TYPE "UDT_CylDiag"
VERSION : 0.1
// -----------------------------------------------------------------------------
// Cylinder Diagnostic - Per-cylinder runtime snapshot
// Used as: DB_Diagnostic.CylDiag[1..8]  (indexed by cylinder number)
// Add new cylinders in OB1 without changing DB_Diagnostic.
// -----------------------------------------------------------------------------
   STRUCT
      State : Int;   // FB_CylinderControl state (-1=EStop 0=Idle 1=Ext... 10=Err)
      Pos : Real;   // Ruler position (mm); 0.0 if no analog sensor connected
      Sol_A : Bool;   // Solenoid A output (extend coil)
      Sol_B : Bool;   // Solenoid B output (retract coil)
      Error : Bool;   // Active error flag
      ErrorID : Word;   // Error code (16#05xx)
   END_STRUCT;

END_TYPE

TYPE "UDT_SpindleSnap"
VERSION : 0.1
// -----------------------------------------------------------------------------
// Spindle Diagnostic Snapshot - one entry in the spindle history ring buffer
// DB_Spindle.Hist_Log[0..19] stores the last 20 state-change events.
// A new entry is pushed whenever SpindleState, PrevStart, ReqStart or StartEdge
// changes value -- so the log captures every meaningful transition without
// flooding with identical scans.
// -----------------------------------------------------------------------------
   STRUCT
      Seq : Int;   // Rolling sequence number
      MachineState : Int;   // FB_Process.State
      State : Int;   // FB_SpindleControl state: 0=Idle 20=Running 30=Halt 999=Error
      ReqStart : Bool;   // FB_RecipeHandler.SpindleReqStart
      ReqStop : Bool;   // FB_RecipeHandler.SpindleReqStop
      bStart : Bool;   // FB_Process bSpindleStart
      bStop : Bool;   // FB_Process bSpindleStop
      StartInput : Bool;   // Composite Start pin at FB_SpindleControl
      StopInput : Bool;   // Composite Stop pin
      EnableIn : Bool;   // bDrivesEnable
      PrevStart : Bool;   // prevStart latch inside FB_SpindleControl
      StartEdge : Bool;   // Rising edge accepted by FB_SpindleControl
      MoveVelBusy : Bool;   // MC_MoveVelocity.Busy  -- TO accepted and processing command
      MoveVelInVel : Bool;   // MC_MoveVelocity.InVelocity -- motor at commanded speed
   END_STRUCT;

END_TYPE

TYPE "AlarmEntry"
VERSION : 0.1
// -----------------------------------------------------------------------------
// Alarm Entry for history
// -----------------------------------------------------------------------------
   STRUCT
      Timestamp {InstructionName := 'DTL'; LibVersion := '1.0'} : DTL;   // RD_SYS_T() at moment of alarm
      ErrorCode : Word;   // 16#xxxx error code
      ProgramNum : Int;   // Active recipe program at fault time (0 = none)
      LineNum : Int;   // Active recipe line at fault time (-1 = outside recipe)
      ErrorText : String[40];   // ITEM-26: English error text snapshot (first 40 chars of DB_HMI.ErrorText)
   END_STRUCT;

END_TYPE

DATA_BLOCK "DB_Error"
{ S7_Optimized_Access := 'TRUE' }
VERSION : 0.1
NON_RETAIN
// DB_ErrorCodes removed -- error codes are used as inline hex constants.
// Severity: 0=info, 1=warn, 2=error, 3=fatal
// -----------------------------------------------------------------------------
// DB_Error - Centralized error snapshot for debugging (non-invasive to HMI)
// -----------------------------------------------------------------------------
   VAR
      Active : Bool;   // TRUE when an active error is present
      Code : Word;   // Error code (matches DB_ErrorCodes)
      Severity : Byte;   // Priority tier: 1=warning, 2=project, 3=motion/TO, 4=safety (higher preempts lower on HMI display)
      Source : String[20];   // Originating FB or category (e.g. 'Recipe', 'Safety')
      Line : Int;   // Recipe line (if applicable) or -1
      TimeStamp {InstructionName := 'DTL'; LibVersion := '1.0'} : DTL;   // Timestamp captured with RD_SYS_T
      Details : String[120];   // Free text details / ActiveErrorText History ring buffer (last 10 errors) for post-mortem analysis
      History_Code : Array[1..10] of Word;
      History_Time {InstructionName := 'DTL'; LibVersion := '1.0'} : Array[1..10] of DTL;
      History_Source : Array[1..10] of String[20];
      History_Details : Array[1..10] of String[80];
      History_Index : Int;   // 1..10
      History_Count : Int;   // Number of valid entries (<=10)
      TotalErrorCount : DInt;   // Lifetime error count (incremented on each new error)
   END_VAR


BEGIN
   Active := FALSE;
   Code := 0;
   Severity := 0;
   Line := -1;
   History_Index := 0;
   History_Count := 0;
   TotalErrorCount := 0;

END_DATA_BLOCK

FUNCTION_BLOCK "FB_Axis_RelPos"
{ S7_Optimized_Access := 'TRUE' }
VERSION : 0.1
// =============================================================================
// FB_Axis_RelPos -- Relative position move (MC_MoveRelative wrapper)
//
// Unlike MC_MoveAbsolute, does not require homing.
// Distance: positive = forward, negative = backward.
// =============================================================================
   VAR_INPUT
      Execute : Bool;
      Distance : Real;   // Relative distance (mm or degrees)
      Velocity : Real;
   END_VAR

   VAR_OUTPUT
      Done : Bool;
      Busy : Bool;
      Error : Bool;
      ErrorID : Word;   // TO error code (MC_MoveRelative.ErrorID)
   END_VAR

   VAR_IN_OUT
      Axis {InstructionName := 'TO_PositioningAxis'; LibVersion := '8.0'} : TO_PositioningAxis;
   END_VAR

   VAR
      MC_MoveRelative_Instance {InstructionName := 'MC_MoveRelative'; LibVersion := '8.0'} : MC_MoveRelative;
      execLatch : Bool;
      prevExec : Bool;
      doneLatch : Bool;
   END_VAR


BEGIN

	IF #Execute AND NOT #prevExec THEN
	    #doneLatch := FALSE;
	    #execLatch := TRUE;
	END_IF;
	#prevExec := #Execute;

	#MC_MoveRelative_Instance(
	                          Axis := #Axis,
	                          Execute := #execLatch,
	                          Distance := #Distance,
	                          Velocity := #Velocity,
	                          Done => #Done,
	                          Busy => #Busy,
	                          Error => #Error
	);
	#ErrorID := #MC_MoveRelative_Instance.ErrorID;

	IF #MC_MoveRelative_Instance.Done OR #MC_MoveRelative_Instance.Error THEN
	    #execLatch := FALSE;
	    #doneLatch := TRUE;
	END_IF;

END_FUNCTION_BLOCK

FUNCTION_BLOCK "FB_Axis_Jog"
{ S7_Optimized_Access := 'TRUE' }
VERSION : 0.1
// =============================================================================
// FB_Axis_Jog -- Continuous jog move
//
// JogForward and JogBackward are level inputs (not edge).
// Axis decelerates when button is released.
// Velocity: jog speed (mm/s) -- fed from DB_Manual.JogSpeed.
// =============================================================================
   VAR_INPUT
      JogForward : Bool;   // Continuous jog in positive direction (level)
      JogBackward : Bool;   // Continuous jog in negative direction (level)
      Velocity : Real;   // Jog speed (mm/s)
   END_VAR

   VAR_OUTPUT
      Busy : Bool;
      Error : Bool;
   END_VAR

   VAR_IN_OUT
      Axis {InstructionName := 'TO_PositioningAxis'; LibVersion := '8.0'} : TO_PositioningAxis;
   END_VAR

   VAR
      MC_MoveJog_Instance {InstructionName := 'MC_MoveJog'; LibVersion := '8.0'} : MC_MoveJog;
   END_VAR


BEGIN

	#MC_MoveJog_Instance(
	                     Axis := #Axis,
	                     JogForward := #JogForward,
	                     JogBackward := #JogBackward,
	                     Velocity := #Velocity,
	                     Busy => #Busy,
	                     Error => #Error
	);

END_FUNCTION_BLOCK

DATA_BLOCK "DB_AlarmHistory"
{ S7_Optimized_Access := 'TRUE' }
VERSION : 0.1
NON_RETAIN
// -----------------------------------------------------------------------------
// DB_AlarmHistory - 20-entry alarm ring buffer for HMI history table (ITEM-26)
// NON_RETAIN: cleared on PLC power cycle. Survives Cmd_Reset (soft reset).
// HMI: connect Hist_Log[0..19] to a table, poll Hist_SeqNum for change detection,
//      sort by Timestamp descending. Hist_Clear = TRUE wipes manually.
// -----------------------------------------------------------------------------
   VAR
      Hist_Head : Int;   // Next write slot (0..19, wraps on overflow)
      Hist_Count : Int;   // Number of valid entries (0..20)
      Hist_SeqNum : DInt;   // Monotonically increasing â€” HMI polls for change detection
      Hist_Clear : Bool;   // HMI writes TRUE to clear history; auto-resets next scan
      Hist_Log : Array[0..19] of "AlarmEntry";
   END_VAR


BEGIN
   Hist_Head := 0;
   Hist_Count := 0;
   Hist_SeqNum := 0;
   Hist_Clear := FALSE;

END_DATA_BLOCK

DATA_BLOCK "DB_HMI_Errors"
{ S7_Optimized_Access := 'TRUE' }
VERSION : 0.1
NON_RETAIN
// -----------------------------------------------------------------------------
// DB_HMI_Errors - Error bits + Word triggers for HMI Alarm View
// -----------------------------------------------------------------------------
// Alarm Words (for HMI Discrete Alarm view)
   VAR
      AlarmWord_Axis : Word;
      AlarmWord_Limits : Word;
      AlarmWord_Tool : Word;
      AlarmWord_Recipe : Word;
      AlarmWord_Safety : Word;
      AlarmWord_Spindle : Word;
      AlarmWord_TO : Word;   // Individual Bool flags
      Err_X_MoveFailed : Bool;
      Err_Z_MoveFailed : Bool;
      Err_X_HomingFailed : Bool;
      Err_Z_HomingFailed : Bool;
      Err_DriveFault : Bool;
      Err_ToolDrivePower : Bool;   // ITEM-29: tool axis drive power fault (error code 0x000D)
      Err_ToolMoveFailed : Bool;
      Err_ToolHomingFailed : Bool;
      Err_MotionTimeout : Bool;
      Err_LockExtendTimeout : Bool;   // 16#0012 -- ToolHeadLock did not confirm engaged within timeout
      Err_SoftLimit_X_Min : Bool;
      Err_SoftLimit_X_Max : Bool;
      Err_SoftLimit_Z_Min : Bool;
      Err_SoftLimit_Z_Max : Bool;
      Err_HWLimit_X_Min : Bool;
      Err_HWLimit_X_Max : Bool;
      Err_HWLimit_Z_Min : Bool;
      Err_HWLimit_Z_Max : Bool;
      Err_InvalidToolNum : Bool;
      Err_ToolOutOfRange : Bool;
      Err_ToolRotTimeout : Bool;
      Err_ToolRetractFail : Bool;
      Err_ToolRotFailed : Bool;
      Err_Recipe_InvalidCmd : Bool;
      Err_Recipe_ParseErr : Bool;
      Err_Recipe_Empty : Bool;
      Err_Recipe_NoLines : Bool;
      Err_PreScan_Limits : Bool;
      Err_Recipe_Feedrate : Bool;
      Err_Recipe_Timeout : Bool;
      Err_Recipe_ToolNum : Bool;
      Err_EStop : Bool;
      Err_EStop_Discrepancy : Bool;   // E-Stop contact discrepancy (channel fault)
      Err_DoorOpen : Bool;
      Err_DrivesNotReady : Bool;
      Err_AirPressure : Bool;
      Err_SafetyInterlock : Bool;
      Err_Spindle_Power : Bool;
      Err_Spindle_Run : Bool;
      Err_Spindle_Halt : Bool;
      Err_Spindle_Speed : Bool;
      Err_TO_Position : Bool;
      Err_TO_Velocity : Bool;
      Err_TO_NotReady : Bool;
      Err_TO_NotEnabled : Bool;
      Err_TO_LimitExceeded : Bool;   // Summary flags
      AnyError : Bool;
      AnySafetyError : Bool;
      AnyAxisError : Bool;
      AnyLimitError : Bool;
      AnyToolError : Bool;
      AnyRecipeError : Bool;
      AnySpindleError : Bool;
   END_VAR


BEGIN

END_DATA_BLOCK

FUNCTION_BLOCK "FB_Axis_Home"
{ S7_Optimized_Access := 'TRUE' }
VERSION : 0.4
// =============================================================================
// FB_Axis_Home -- Homing
//
// Mode options (MC_Home Mode parameter):
//   0 -- Passive: only set current position to Position value
//   2 -- Active:  go to reference switch, zero encoder
//   3 -- Active + Zero: go to reference switch, set Position value
//
// Default mode = 3 (matches DB_Manual.HomingMode).
//
// Safety note: Execute is rising-edge triggered -- even if Execute stays TRUE
// after Done/Error, a new homing will not start. Same pattern as FB_Axis_AbsPos.
// =============================================================================
   VAR_INPUT
      Execute : Bool;   // Rising edge = start homing
      Mode : Int := 3;   // Homing mode (0=Passive, 2=Active, 3=Active+Zero)
      Position : Real := 0.0;   // Position value after homing (usually 0.0)
   END_VAR

   VAR_OUTPUT
      Done : Bool;
      Busy : Bool;
      Error : Bool;
      ErrorID : Word;   // MC_Home TO error code -- converted to readable text via FC_TO_ErrorText
   END_VAR

   VAR_IN_OUT
      Axis {InstructionName := 'TO_PositioningAxis'; LibVersion := '8.0'} : TO_PositioningAxis;
   END_VAR

   VAR
      MC_Home_Instance {InstructionName := 'MC_Home'; LibVersion := '8.0'} : MC_Home;
      execInternal : Bool;   // Actual Execute sent to MC_Home
      prevExecute : Bool;   // Previous Execute value for edge detection
      doneLatch : Bool;   // Prevents re-trigger after Done/Error
   END_VAR


BEGIN

	// Rising edge: new command -- clear doneLatch
	IF #Execute AND NOT #prevExecute THEN
	    #doneLatch := FALSE;
	END_IF;
	#prevExecute := #Execute;

	// execInternal: run if new command and not yet done, OR still busy
	// This ensures Execute staying TRUE after Done does not restart homing
	#execInternal := (#Execute AND NOT #doneLatch) OR #MC_Home_Instance.Busy;

	#MC_Home_Instance(
	                  Axis := #Axis,
	                  Execute := #execInternal,
	                  Position := #Position,
	                  Mode := #Mode,
	                  Done => #Done,
	                  Busy => #Busy,
	                  Error => #Error
	);

	// Done or Error: set doneLatch -- cannot re-trigger without Execute FALSEâ†’TRUE
	IF #MC_Home_Instance.Done OR #MC_Home_Instance.Error THEN
	    #doneLatch := TRUE;
	END_IF;

	// Pass TO error code out -- written to DB_Diagnostic in FB_Process
	#ErrorID := #MC_Home_Instance.ErrorID;

END_FUNCTION_BLOCK

TYPE "RecipeHeader"
VERSION : 0.1
   STRUCT
      sName : String[20];   // Program name (max 20 chars)
      LineCount : Int;   // Total lines in program (0-999)
      Valid : Bool;   // Program is valid and loaded
      PreScanned : Bool;   // Pre-scan completed
      MinX : Real;   // Bounding box Min X
      MaxX : Real;   // Bounding box Max X
      MinZ : Real;   // Bounding box Min Z
      MaxZ : Real;   // Bounding box Max Z
   END_STRUCT;

END_TYPE

DATA_BLOCK "DB_ToolConfig"
{ S7_Optimized_Access := 'TRUE' }
VERSION : 0.2
NON_RETAIN
// -----------------------------------------------------------------------------
// DB_ToolConfig - Tool changer configuration
// -----------------------------------------------------------------------------
// Slot angles -- automatically calculated by FC_ToolAngleCalc (AutoCalcAngles=TRUE)
// or manually entered from HMI Tool page (AutoCalcAngles=FALSE).
   VAR
      Tool1_Position : Real;   // Slot 1 angle (degrees)
      Tool2_Position : Real;   // Slot 2 angle (degrees)
      Tool3_Position : Real;   // Slot 3 angle (degrees)
      Tool4_Position : Real;   // Slot 4 angle (degrees) Slot code mapping -- can be entered from HMI Tool page. Operator enters which head code is in which slot.
      ToolCode_List : Array[1..4] of Int;
      CurrentTool : Int;   // Active slot number (1-4) HMI Tool page: automatic angle calculation TRUE = calculate evenly spaced based on ToolCount (e.g. 4 slots â†’ 0/90/180/270) FALSE = Tool1..4_Position open for manual entry
      AutoCalcAngles : Bool;   // Calculated step angle -- displayed on HMI for information (e.g. "90Â°/slot")
      ToolStepAngle_Calc : Real;
   END_VAR


BEGIN
   Tool1_Position := 0.0;
   Tool2_Position := 120.0;
   Tool3_Position := 240.0;
   Tool4_Position := 360.0;
   ToolCode_List[1] := 101;
   ToolCode_List[2] := 102;
   ToolCode_List[3] := 103;
   ToolCode_List[4] := 104;
   CurrentTool := 1;
   AutoCalcAngles := TRUE;
   ToolStepAngle_Calc := 120.0;

END_DATA_BLOCK

DATA_BLOCK "DB_MachineConfig"
{ S7_Optimized_Access := 'TRUE' }
VERSION : 0.2
NON_RETAIN
// -----------------------------------------------------------------------------
// DB_MachineConfig - Machine configuration parameters
// -----------------------------------------------------------------------------
// =====================================================================
// HMI-EDITABLE: Machine Physical Limits (mm)
// These values are NOT overwritten by FC_LoadConfig.
// Can be changed from HMI Setup screen; preserved on PLC restart.
// =====================================================================
   VAR
      SoftLimit_MinX : Real;   // X minimum (home=0)
      SoftLimit_MaxX : Real;   // X maximum travel (mm)
      SoftLimit_MinZ : Real;   // Z minimum (negative = mandrel front / clearance)
      SoftLimit_MaxZ : Real;   // Z maximum (forming depth) HMI-EDITABLE: Safe Positions (mm)
      SafePos_X : Real;   // "Go Safe" X target
      SafePos_Z : Real;   // "Go Safe" Z target (clearance zone) HMI-EDITABLE: Pause Retract (mm / mm/s) On Pause, X and Z jog by these signed offsets to pull the tool clear (spindle keeps running). On Continue they return to the exact interruption point before the recipe resumes. Retract target is clamped to soft limits. Offset 0 = that axis does not move on pause. See docs/Pause_Retract_Plan.md.
      PauseRetract_X : Real;   // Pause retract offset X (signed, mm)
      PauseRetract_Z : Real;   // Pause retract offset Z (signed, mm)
      PauseRetract_Vel : Real;   // Retract/return velocity (mm/s) HMI-EDITABLE: Homing Parameters
      HomeOffset_X : Real;   // X set value after homing
      HomeOffset_Z : Real;   // Z set value after homing
      HomeVelocity : Real;   // Homing clearance velocity (mm/s)
      PostHome_Clearance : Real;   // Distance to clear PNP zone after homing (mm)
      AlwaysHomeOnAutoStart : Bool;   // TRUE = home all axes on every auto start (recommended) âš ï¸ UNUSED: The following two parameters are not read anywhere in PLC code. Recipe handler takes its own feedrate from the recipe line. Do not connect to HMI. May be used if manual tool change sequence is added later.
      ToolChangePos_X : Real;   // (Unused) Safe X for manual tool change
      ToolChangePos_Z : Real;   // (Unused) Safe Z for manual tool change
      DefaultFeedrate : Real;   // (Unused) Default feedrate ===================================================================== FIXED: Hardware/TO Limits -- must not be changed from HMI FC_LoadConfig (OB100) writes these values on every restart. =====================================================================
      MaxVelocity : Real;   // mm/s - TO max velocity
      RapidVelocity : Real;   // mm/s - G0 rapid speed
      MinVelocity : Real;   // mm/s - TO minimum
      FeedrateConvFactor : Real;   // divisor to convert recipe F (mm/min) to axis velocity (mm/s) Tool Configuration -- HMI-EDITABLE: active slot count (1-4)
      ToolCount : Int;
      ToolVelocity : Real;   // deg/s -- turret rotation speed (clamped by TO max) Hardware configuration -- set TRUE if this axis is not physically connected to the machine (different from HMI bypasses: this is a hardware presence flag)
      Bypass_ToolAxis : Bool;
      Bypass_MandrelLock : Bool;   // Spindle deceleration wait: time between RunCmd=FALSE and next RunCmd=TRUE. Set to match VFD deceleration ramp time. HMI-editable.
      SpindleDecelTime : Time;   // Proportional MandrelLock release wait (ITEM-28). SpindleStopSafeTime = full-speed stop safety margin (tune to measured VFD decel time + margin). Formula: PT = (capturedRPM / SpindleMaxRPM) * SpindleStopSafeTime
      SpindleMaxRPM : Real;   // RPM -- denominator for proportional wait (match DB_Spindle.MaxSpeed)
      SpindleStopSafeTime : Time;   // Full-speed decel safety margin (tune on-site) â”€â”€â”€ Cylinder stroke wait times (open-loop: tuned to physical stroke duration) These are deliberate waits with no sensor feedback. Set slightly above measured stroke time.
      CylMandrelLock_ClampTime : Time;   // STATE_SHEET_WAIT ph.2: MandrelLock clamp stroke
      CylSheetHolder_RetractTime : Time;   // STATE_SHEET_WAIT ph.3: SheetHolder retract stroke
      CylToolHeadLock_PreDelay : Time;   // STATE_LOCK_EXTEND_WAIT: pre-delay before solenoid energises
      CylToolHeadLock_RetractTime : Time;   // STATE_LOCK_RETRACT_WAIT: spring-return wait (no sensor) â”€â”€â”€ Process timeouts (trigger errors when limits exceeded)
      Timeout_DriveReady : Time;   // STATE_STARTING: drives not ready within this time â†’ error
      Timeout_Homing : Time;   // STATE_HOMING + STATE_STOP_GOHOME combined timeout
      Timeout_Motion : Time;   // Per-line G0/G1 motion timeout in FB_RecipeHandler
      Timeout_SpindleAtSpeed : Time;   // CMD=20: spindle must reach target speed within this time
      Timeout_SpindleStop : Time;   // CMD=21: spindle must reach zero within this time
      Timeout_ToolChange : Time;   // Turret rotation must complete within this time
      Timeout_EStopDiscrep : Time;   // E-Stop dual-channel discrepancy debounce
   END_VAR


BEGIN
   SoftLimit_MinX := -10.0;
   SoftLimit_MaxX := 500.0;
   SoftLimit_MinZ := -10.0;
   SoftLimit_MaxZ := 500.0;
   SafePos_X := 0.0;
   SafePos_Z := 0.0;
   PauseRetract_X := -10.0;
   PauseRetract_Z := -10.0;
   PauseRetract_Vel := 30.0;
   HomeOffset_X := 0.0;
   HomeOffset_Z := 0.0;
   HomeVelocity := 10.0;
   PostHome_Clearance := 10.0;
   AlwaysHomeOnAutoStart := TRUE;
   ToolChangePos_X := 0.0;
   ToolChangePos_Z := 0.0;
   DefaultFeedrate := 100.0;
   MaxVelocity := 40.0;
   RapidVelocity := 40.0;
   MinVelocity := 1.0;
   FeedrateConvFactor := 60.0;
   ToolCount := 3;
   ToolVelocity := 50.0;
   Bypass_ToolAxis := FALSE;
   Bypass_MandrelLock := FALSE;
   SpindleDecelTime := T#2S;
   SpindleMaxRPM := 2400.0;
   SpindleStopSafeTime := T#20S;
   CylMandrelLock_ClampTime := T#5S;
   CylSheetHolder_RetractTime := T#5S;
   CylToolHeadLock_PreDelay := T#1S;
   CylToolHeadLock_RetractTime := T#3S;
   Timeout_DriveReady := T#3S;
   Timeout_Homing := T#2M;
   Timeout_Motion := T#5M;
   Timeout_SpindleAtSpeed := T#10S;
   Timeout_SpindleStop := T#15S;
   Timeout_ToolChange := T#30S;
   Timeout_EStopDiscrep := T#500MS;

END_DATA_BLOCK

FUNCTION_BLOCK "FB_Axis_Halt"
{ S7_Optimized_Access := 'TRUE' }
VERSION : 0.2
// =============================================================================
// FB_Axis_Halt -- Controlled stop
//
// Execute = TRUE â†’ MC_Halt called, axis decelerates to a stop.
// Cancels any active MC_MoveAbsolute.
// Done = TRUE â†’ axis has fully stopped.
// =============================================================================
   VAR_INPUT
      Execute : Bool;   // TRUE = issue stop command
   END_VAR

   VAR_OUTPUT
      Done : Bool;
      Busy : Bool;
      Error : Bool;
      ErrorID : Word;   // MC_Halt TO error code -- available for diagnostics on halt failure
   END_VAR

   VAR_IN_OUT
      Axis {InstructionName := 'TO_PositioningAxis'; LibVersion := '8.0'} : TO_PositioningAxis;
   END_VAR

   VAR
      MC_Halt_Instance {InstructionName := 'MC_Halt'; LibVersion := '8.0'} : MC_Halt;
   END_VAR


BEGIN

	#MC_Halt_Instance(
	                  Axis := #Axis,
	                  Execute := #Execute,
	                  Done => #Done,
	                  Busy => #Busy,
	                  Error => #Error,
	                  ErrorID => #ErrorID
	);

END_FUNCTION_BLOCK

TYPE "RecipeLine"
VERSION : 0.1
   STRUCT
      X : Real;   // 4 bytes - Target X position (mm)
      Z : Real;   // 4 bytes - Target Z position (mm)
      F : Int;   // 2 bytes - Feedrate (mm/min, 0=rapid)
      CMD : Byte;   // 1 byte  - Command: 0=G0, 1=G1, 10=Tool, 20=SpindleOn, 21=SpindleOff, 30=Dwell, 99=End
      Param : Byte;   // 1 byte  - CMD=10:ToolNum, CMD=20:RPM/10, CMD=30:Time*100ms
   END_STRUCT;

END_TYPE

DATA_BLOCK "DB_HMI"
{ S7_Optimized_Access := 'TRUE' }
VERSION : 0.3
NON_RETAIN
// =============================================================================
// 02_DataBlocks.scl
// All non-recipe data blocks.
// Recipe program DBs (DB_RecipeProgram1..5) are in 02b_RecipePrograms.scl.
// Target: CPU 1214C (100KB work memory)
// =============================================================================
// -----------------------------------------------------------------------------
// DB_HMI - Human Machine Interface data
// -----------------------------------------------------------------------------
// ===========================================================
// BUTTONS (Input) - Version_GCODE compatible
// ===========================================================
   VAR
      Btn_Start : Bool;   // Start machine
      Btn_Stop : Bool;   // Stop machine
      Btn_Pause : Bool;   // Pause/Resume toggle
      Btn_Reset : Bool;   // Reset program to beginning
      Btn_ApplyToolConfig : Bool;   // Apply tool-slot codes from HMI to DB_ToolConfig
      Btn_AckError : Bool;   // Acknowledge error â†’ transitions from STATE_ERROR to STOPPED
      Btn_Continue : Bool;   // Continue from pause (PAUSED) -- STATE_PAUSED â†’ RUNNING
      Btn_Restart : Bool;   // STATE_ERROR or PAUSED â†’ STOPPED (restart with Start)
      Btn_ProdReset : Bool;   // Reset production counters + history
      Btn_LastCycleReset : Bool;   // Reset last cycle summary only (counters preserved) NOTE: Btn_ProdReset already does this too. If not adding both as separate HMI buttons, Btn_LastCycleReset is redundant -- do not connect to HMI if unused. =========================================================== MODE SELECTION (Input) ===========================================================
      ProductSelect : Int;   // Recipe selector (1-5)
      FeedrateOverride : Real;   // Speed % for G1 moves (50-200, 100=normal)
      RapidOverride : Real;   // Speed % for G0 rapid moves (50-200)
      SingleStepMode : Bool;   // TRUE = stop after each line, wait for StepNext
      StepNext : Bool;   // Pulse to advance one step in SingleStepMode Program names and validity -- PLC does NOT write to these tags. Written by CAM post-processor or HMI operator. Can be read for displaying the program list on HMI.
      ProgramNames : Array[1..5] of String[20];   // Operator-defined program names
      ProgramValid : Array[1..5] of Bool;   // Is program loaded? (written by HMI/CAM) Tool slot codes editable from HMI. Enter external codes like 101, 406 etc. These are copied to DB_ToolConfig.ToolCode_List when operator presses Apply.
      ToolSlotCode : Array[1..4] of Int;   // =========================================================== POSITION DISPLAYS (Output) ===========================================================
      ActualX : Real;   // Current X position (mm)
      ActualZ : Real;   // Current Z position (mm) =========================================================== STATUS DISPLAYS (Output) ===========================================================
      StatusMsg : String[50];   // Status message text
      MachineState : Int;   // State machine state
      CurrentLine : Int;   // Current line being executed
      TotalLines : Int;   // Total lines in program
      ProgressPercent : Real;   // Progress 0-100%
      CurrentTool : Int;   // Active tool (1-4)
      FeedrateActive : Real;   // Actual feedrate (mm/min) âš ï¸ UNUSED: PLC code does not write to the Axis_Status_* tags below anywhere. They will always be 0 / empty if connected to HMI. Reserved for future use -- do not display on HMI for now.
      Axis_Status_X : Int;
      Axis_Status_Z : Int;
      Axis_Status_Spindle : Int;
      Axis_Status_Toolhead : Int;
      Axis_Status_X_Str : String[10];
      Axis_Status_Z_Str : String[10];
      Axis_Status_Spindle_Str : String[10];
      Axis_Status_Toolhead_Str : String[10];   // =========================================================== STATUS LAMPS (Output) ===========================================================
      IsRunning : Bool;   // Machine is running
      IsPaused : Bool;   // Machine is paused
      HasError : Bool;   // Error is active
      ElapsedTime : Time;   // Program elapsed time
      ElapsedSeconds : DInt;   // Elapsed time in seconds (for HMI display)
      CycleCount : Int;   // Number of completed programs =========================================================== ERROR DISPLAY (Output) ===========================================================
      ErrorID : Word;   // Error code (0=OK)
      ErrorText : String[100];   // Error description
      ErrorDetail : String[120];   // Additional error info =========================================================== WARNING DISPLAY (Output) ===========================================================
      HasWarning : Bool;   // TRUE when a non-blocking warning is active (E-Stop bypass or sheet insert prompt)
      WarningText : String[70];   // Warning message text -- English (E-Stop bypass or operator prompts only)
      ResumeLine : Int;   // Saved recipe line for warm restart (-1 = none). Set in STATE_ERROR, cleared on Btn_Restart. =========================================================== SPANISH TEXT MIRRORS (Output) -- for Mexican operator HMI PLC writes these every scan alongside the English equivalents. Connect to a second-language screen or a language-toggle switch. ===========================================================
      StatusMsg_ES : String[50];   // Estado actual (EspaÃ±ol)
      ErrorText_ES : String[100];   // Descripcion de error (EspaÃ±ol)
      ErrorDetail_ES : String[120];   // Detalle adicional (EspaÃ±ol)
      WarningText_ES : String[80];   // Advertencia (EspaÃ±ol) =========================================================== BYPASS SWITCHES (for testing) - Version_GCODE compatible âš ï¸ All bypasses reset to FALSE on restart (FC_LoadConfig). All must be FALSE in production. ===========================================================
      Bypass_EStop : Bool;   // Used in FB_SafetyMonitor âœ…
      Bypass_Door : Bool;   // Used in FB_SafetyMonitor âœ…
      Bypass_AirPressure : Bool;   // Used in FB_SafetyMonitor âœ…
      Bypass_Drives : Bool;   // Used in FB_SafetyMonitor âœ…
      Bypass_Spindle : Bool;   // Skips spindle commands in recipe (FB_RecipeHandler) -- dry run / commissioning
      Bypass_ToolChanger : Bool;   // âš ï¸ UNUSED -- not in safety monitor
      Bypass_MandrelLock : Bool;   // TRUE = machine variant without MandrelLock cylinder (manual clamping) =========================================================== BOUNDING BOX (Output - from pre-scan) ===========================================================
      BoundingBox_MinX : Real;
      BoundingBox_MaxX : Real;
      BoundingBox_MinZ : Real;
      BoundingBox_MaxZ : Real;
      BoundingBox_Valid : Bool;
      PreScanProgress : Real;   // Pre-scan progress 0-100% (written during STATE_PRE_SCAN) =========================================================== MANUAL > MANAGE: Contactor & Enable controls (Input) HMI writes these; PLC drives physical outputs in OB1. Buttons are toggles (maintained, not momentary). ===========================================================
      Btn_Contactor_X : Bool;   // Energize X driver contactor
      Btn_Contactor_Z : Bool;   // Energize Z driver contactor
      Btn_Contactor_Tool : Bool;   // Energize Tool driver contactor
      Btn_Contactor_Spindle : Bool;   // Energize Spindle driver contactor
      Btn_Enable_X : Bool;   // Send enable signal to X drive
      Btn_Enable_Z : Bool;   // Send enable signal to Z drive MANUAL > MANAGE: Status feedback (Output) for HMI lamps PLC writes these back after applying safety interlock.
      Contactor_X_On : Bool;
      Contactor_Z_On : Bool;
      Contactor_Tool_On : Bool;
      Contactor_Spindle_On : Bool;
      Enable_X_On : Bool;
      Enable_Z_On : Bool;   // =========================================================== E-STOP DUAL CHANNEL STATUS (Output - PLC writes, HMI reads) ===========================================================
      EStop_Ch1_OK : Bool;   // Channel 1 contact state (TRUE=closed=safe)
      EStop_Ch2_OK : Bool;   // Channel 2 contact state (TRUE=closed=safe)
      EStop_Discrepancy : Bool;   // Ch1 â‰  Ch2 â†’ contact fault, service required
   END_VAR


BEGIN
   ProductSelect := 1;
   FeedrateOverride := 100.0;
   RapidOverride := 100.0;
   SingleStepMode := FALSE;
   StepNext := FALSE;
   ToolSlotCode[1] := 101;
   ToolSlotCode[2] := 102;
   ToolSlotCode[3] := 103;
   ToolSlotCode[4] := 104;
   ResumeLine := -1;
   Bypass_EStop := FALSE;
   Bypass_Door := TRUE;
   Bypass_AirPressure := TRUE;
   Bypass_Drives := FALSE;
   Bypass_Spindle := FALSE;
   Bypass_ToolChanger := FALSE;
   Bypass_MandrelLock := FALSE;
   PreScanProgress := 0.0;

END_DATA_BLOCK

DATA_BLOCK "DB_Diagnostic"
{ S7_Optimized_Access := 'TRUE' }
VERSION : 0.1
NON_RETAIN
// -----------------------------------------------------------------------------
// DB_Diagnostic - Runtime diagnostics and debugging
// -----------------------------------------------------------------------------
// =========================================================
// PROCESS STATE
// =========================================================
   VAR
      Process_State : Int;
      Process_SafeToRun : Bool;
      Process_DrivesEnable : Bool;   // ========================================================= RECIPE HANDLER STATE =========================================================
      Recipe_CurrentProgram : Int;   // Active program number (1-5)
      Recipe_CurrentLine : Int;   // Current line being executed
      Recipe_TotalLines : Int;   // Total lines in program
      Recipe_TargetX : Real;   // Current target X
      Recipe_TargetZ : Real;   // Current target Z
      Recipe_Velocity : Real;   // Current velocity Pre-scan results
      PreScan_Complete : Bool;
      PreScan_Valid : Bool;   // No limit violations found
      PreScan_ErrorLine : Int;   // Line with limit error (-1 if none) ========================================================= MOVE STATUS =========================================================
      MoveX_Busy : Bool;
      MoveX_Done : Bool;
      MoveX_Error : Bool;
      MoveZ_Busy : Bool;
      MoveZ_Done : Bool;
      MoveZ_Error : Bool;
      bMoveX : Bool;   // X axis needs to move
      bMoveZ : Bool;   // Z axis needs to move ========================================================= AXIS INFO (commissioning) =========================================================
      Axis_X_Pos : Real;
      Axis_Z_Pos : Real;
      Axis_X_Enabled : Bool;
      Axis_Z_Enabled : Bool;
      Axis_X_Homed : Bool;
      Axis_Z_Homed : Bool;   // ========================================================= ERROR CONTEXT =========================================================
      Error_ProcessState : Int;
      Error_Line : Int;
      Error_Code : Word;   // TO error codes -- raw WORD codes from Siemens MC_ function blocks. Converted to readable text via FC_TO_ErrorText; compare with TIA Portal TO Diagnostics.
      MoveX_ErrorID : Word;   // MC_MoveAbsolute X axis TO code
      MoveZ_ErrorID : Word;   // MC_MoveAbsolute Z axis TO code
      HomeX_ErrorID : Word;   // MC_Home X axis TO code
      HomeZ_ErrorID : Word;   // MC_Home Z axis TO code
      HomeTool_ErrorID : Word;   // MC_Home Tool axis TO code
      Power_X_ErrorID : Word;   // MC_Power X axis TO code
      Power_Z_ErrorID : Word;   // MC_Power Z axis TO code
      Spindle_TO_ErrorID : Word;   // MC_Power/MC_MoveVelocity/MC_Halt spindle TO code
      Error_Text : String[100];   // Error_Detail removed -- not written anywhere, Error_Text is used instead Readable description for the last TO error code (FC_TO_ErrorText output)
      TO_ErrorText : String[60];   // ========================================================= CYLINDER DIAGNOSTICS -- indexed by cylinder number (1-based, max 8) No new fields needed when adding cylinders -- write to CylDiag[N] in OB1. =========================================================
      CylDiag : Array[1..8] of "UDT_CylDiag";
   END_VAR


BEGIN

END_DATA_BLOCK

DATA_BLOCK "DB_Spindle"
{ S7_Optimized_Access := 'TRUE' }
VERSION : 0.2
NON_RETAIN
// -----------------------------------------------------------------------------
// DB_Spindle - Spindle configuration and status
// -----------------------------------------------------------------------------
// Configuration
   VAR
      MinSpeed : Real;   // Minimum spindle speed (RPM)
      MaxSpeed : Real;   // Maximum spindle speed (RPM)
      DefaultSpeed : Real;   // Default spindle speed (RPM)
      SpeedTolerance : Real;   // Speed tolerance for AtSpeed (%)
      Bypass_AtSpeed : Bool;   // TRUE = skip AtSpeed wait (use during commissioning without drive) Commands (input from HMI/Program)
      Cmd_SetSpeed : Real;   // Commanded speed
      Cmd_Direction : Int;   // 1=CW, -1=CCW
      SpeedOverride : Real;   // Speed override (%) Status (output)
      IsRunning : Bool;
      AtSpeed : Bool;
      ActualSpeed : Real;
      CommandedSpeed : Real;
      Error : Bool;
      ErrorID : Word;   // ===================================================================== DIAGNOSTICS -- written every scan; read from HMI watch table Use these to trace the spindle start chain without TIA Portal online. Chain:  ReqStart â†’ bSpindleStart â†’ StartInput â†’ PrevStart â†’ StartEdge â†’ state =====================================================================
      Diag_SpindleState : Int;   // FB_SpindleControl state (0=Idle, 10=Starting, 20=Running, 30=Stopping, 999=Error)
      Diag_StartInput : Bool;   // Actual Start pin arriving at FB_SpindleControl (Manual OR bSpindleStart)
      Diag_StopInput : Bool;   // Actual Stop pin arriving at FB_SpindleControl
      Diag_EnableInput : Bool;   // Actual Enable pin (bDrivesEnable)
      Diag_StartEdge : Bool;   // Rising edge computed inside FB_SpindleControl (TRUE = spindle command accepted)
      Diag_PrevStart : Bool;   // prevStart latch inside FB_SpindleControl (must go FALSE between starts)
      Diag_bSpindleStart : Bool;   // FB_Process internal flag bSpindleStart (set by recipe or RUNNING state)
      Diag_bSpindleStop : Bool;   // FB_Process internal flag bSpindleStop
      Diag_ReqStart : Bool;
      Diag_ReqStop : Bool;
      Diag_MoveVelBusy : Bool;   // MC_MoveVelocity.Busy   -- TO is processing the velocity command
      Diag_MoveVelInVel : Bool;   // MC_MoveVelocity.InVelocity -- motor reached commanded speed ===================================================================== HISTORY RING BUFFER -- last 20 state-change snapshots A new entry is pushed whenever SpindleState, PrevStart, ReqStart or StartEdge changes, capturing every meaningful transition in sequence. How to read:   1. Hist_Count tells you how many valid entries exist (0..20).   2. Hist_Head-1 (mod 20) is the MOST RECENT entry.   3. Entries are indexed [0..19]; read them in Seq order.   4. Write Hist_Clear := TRUE from HMI to wipe and start fresh. =====================================================================
      Hist_Head : Int;   // Next write position (0..19, wraps)
      Hist_Count : Int;   // Number of valid entries (0..20)
      Hist_SeqNum : Int;   // Rolling sequence counter
      Hist_Clear : Bool;   // HMI: write TRUE to clear buffer (auto-resets)
      Hist_Log : Array[0..19] of "UDT_SpindleSnap";
   END_VAR


BEGIN
   MinSpeed := 120.0;
   MaxSpeed := 3000.0;
   DefaultSpeed := 1200.0;
   SpeedTolerance := 5.0;
   Bypass_AtSpeed := FALSE;
   SpeedOverride := 100.0;
   IsRunning := FALSE;
   AtSpeed := FALSE;
   ActualSpeed := 0.0;
   CommandedSpeed := 0.0;
   Error := FALSE;
   ErrorID := 0;
   Hist_Head := 0;
   Hist_Count := 0;
   Hist_SeqNum := 0;
   Hist_Clear := FALSE;

END_DATA_BLOCK

DATA_BLOCK "DB_SystemEvents"
{ S7_Optimized_Access := 'TRUE' }
VERSION : 0.2
NON_RETAIN
// =============================================================================
// Version_Recipe - 07_ReportError.scl
// Central helper to report errors from any FB/FC/FCU without duplicating logic.
// =============================================================================
// ---------------------------------------------------------------------------
// DB_SystemEvents - small DB for inter-block requests (error reporting)
// ---------------------------------------------------------------------------
// Error queue: ring buffer (4 slots) -- prevents silent loss when two errors
// occur in the same scan before FB_AlarmManager can consume the first entry.
// FC_ReportError enqueues; FB_AlarmManager dequeues one item per scan.
   VAR
      EQ_Head : Int;   // Next slot to dequeue (read index)
      EQ_Tail : Int;   // Next slot to enqueue (write index)
      EQ_Count : Int;   // Number of pending items (0..4)
      EQ_Code : Array[0..3] of Word;
      EQ_Details : Array[0..3] of String[80];
      EQ_Source : Array[0..3] of String[20];
   END_VAR


BEGIN
   EQ_Head := 0;
   EQ_Tail := 0;
   EQ_Count := 0;

END_DATA_BLOCK

FUNCTION_BLOCK "FB_Axis_AbsPos"
{ S7_Optimized_Access := 'TRUE' }
VERSION : 1.0
// =============================================================================
// 03_AxisControl.scl
// Axis control wrapper function blocks
//
// This file wraps Siemens PLCopen MC_ commands with project-specific thin wrappers.
// All FBs accept a TO_PositioningAxis VAR_IN_OUT reference.
//
// FB List:
//   FB_Axis_AbsPos  -- Absolute position move (MC_MoveAbsolute wrapper)
//   FB_Axis_Power   -- Drive enable/disable (MC_Power wrapper)
//   FB_Axis_Home    -- Homing (MC_Home wrapper)
//   FB_Axis_Halt    -- Controlled stop (MC_Halt wrapper)
//   FB_Axis_Jog     -- Continuous jog (MC_MoveJog wrapper)
//   FB_Axis_Reset   -- TO error reset (MC_Reset wrapper)
//
// Units: mm and mm/s (must match Technology Object configuration).
// =============================================================================
// =============================================================================
// FB_Axis_AbsPos -- Absolute position move
//
// Behavior:
//   Starts a new move on the rising edge of Execute.
//   Done = TRUE remains set while Execute is TRUE after completion.
//   Clearing Execute also clears Done -- ready for the next command.
//
// Usage note:
//   Used by FB_RecipeHandler and FB_ManualMode.
//   Two simultaneous Execute signals must not be sent to the same axis.
// =============================================================================
   VAR_INPUT
      Execute : Bool;   // Rising edge = new move command
      Position : Real;   // Target position (mm)
      Velocity : Real;   // Move velocity (mm/s)
   END_VAR

   VAR_OUTPUT
      Done : Bool;   // Move completed
      Busy : Bool;   // Move in progress
      Error : Bool;   // TO/drive error
      ErrorID : Word;   // MC_ error code (compare with TO diagnostics)
   END_VAR

   VAR_IN_OUT
      Axis {InstructionName := 'TO_PositioningAxis'; LibVersion := '8.0'} : TO_PositioningAxis;
   END_VAR

   VAR
      MC_MoveAbsolute_Instance {InstructionName := 'MC_MoveAbsolute'; LibVersion := '8.0'} : MC_MoveAbsolute;
      execLatch : Bool;   // MC_MoveAbsolute Execute latch -- ensures single command
      doneLatch : Bool;   // Holds Done result until Execute goes FALSE
      prevExecute : Bool;   // Previous Execute value for edge detection
   END_VAR


BEGIN

	// Rising edge: new command starting -- clear previous Done
	IF #Execute AND NOT #prevExecute THEN
	    #doneLatch := FALSE;
	END_IF;
	#prevExecute := #Execute;

	// If Execute is active, not yet done, and latch not set -- start move
	IF #Execute AND NOT #execLatch AND NOT #doneLatch THEN
	    #execLatch := TRUE;
	END_IF;

	// MC_MoveAbsolute call
	#MC_MoveAbsolute_Instance(
	                          Axis := #Axis,
	                          Execute := #execLatch,
	                          Position := #Position,
	                          Velocity := #Velocity,
	                          Done => #Done,
	                          Busy => #Busy,
	                          Error => #Error,
	                          ErrorID => #ErrorID
	);

	// Done: release latch, hold done result
	IF #MC_MoveAbsolute_Instance.Done THEN
	    #execLatch := FALSE;
	    #doneLatch := TRUE;
	    // Error or CommandAborted: release latch, do NOT set doneLatch
	    // CommandAborted happens when MC_Halt interrupts a running move (stop/pause/reset).
	    // Without this branch execLatch stays TRUE across recipe runs, MC never gets a new
	    // rising edge on Execute, and the axis stands still on the next start.
	ELSIF #MC_MoveAbsolute_Instance.Error OR #MC_MoveAbsolute_Instance.CommandAborted THEN
	    #execLatch := FALSE;
	END_IF;

	// Done: latch or MC instant done -- visible while Execute is TRUE
	#Done := #doneLatch OR #MC_MoveAbsolute_Instance.Done;
	#Error := #MC_MoveAbsolute_Instance.Error;

END_FUNCTION_BLOCK

FUNCTION_BLOCK "FB_InputManager"
{ S7_Optimized_Access := 'TRUE' }
VERSION : 1.0
// =============================================================================
// Version_Recipe - 06_MainProcess.scl
// Main process with recipe-based G-code and pre-scan validation
// =============================================================================
// -----------------------------------------------------------------------------
// FB_InputManager - OR-combine inputs from HMI, Panel, Remote
// DOC:
//  purpose: Create single rising-edge command outputs (Cmd_*) from multiple input sources.
//  inputs: HMI_*, Panel_*, Rem_* (Bool) - raw button states (level)
//  outputs: Cmd_* (Bool) - one-shot rising-edge commands for the system
//  notes: Uses prev* latches to detect rising edges; keeps logic simple for deterministic behavior.
// -----------------------------------------------------------------------------
   VAR_INPUT
      HMI_Start : Bool;   // HMI Start button (level)
      HMI_Stop : Bool;   // HMI Stop button (level)
      HMI_Pause : Bool;   // HMI Pause button (level)
      HMI_Reset : Bool;   // HMI Reset button (level)
      Panel_Start : Bool;   // Physical panel Start
      Panel_Stop : Bool;   // Physical panel Stop
      Panel_Pause : Bool;   // Physical panel Pause
      Panel_Reset : Bool;   // Physical panel Reset
      Rem_Start : Bool;   // Remote Start (e.g. PLC network)
      Rem_Stop : Bool;   // Remote Stop One-shot command outputs (rising edge true for one cycle)
   END_VAR

   VAR_OUTPUT
      Cmd_Start : Bool;
      Cmd_Stop : Bool;
      Cmd_Pause : Bool;
      Cmd_Reset : Bool;   // Previous sampled raw values for edge detection
   END_VAR

   VAR
      prevStart : Bool;
      prevStop : Bool;
      prevPause : Bool;
      prevReset : Bool;   // Combined raw inputs for current cycle
      rawStart : Bool;
      rawStop : Bool;
      rawPause : Bool;
      rawReset : Bool;
   END_VAR


BEGIN

	#rawStart := #HMI_Start OR #Panel_Start OR #Rem_Start;
	#rawStop := #HMI_Stop OR #Panel_Stop OR #Rem_Stop;
	#rawPause := #HMI_Pause OR #Panel_Pause;
	#rawReset := #HMI_Reset OR #Panel_Reset;
	#Cmd_Start := #rawStart AND NOT #prevStart;
	#Cmd_Stop := #rawStop AND NOT #prevStop;
	#Cmd_Pause := #rawPause AND NOT #prevPause;
	#Cmd_Reset := #rawReset AND NOT #prevReset;
	#prevStart := #rawStart;
	#prevStop := #rawStop;
	#prevPause := #rawPause;
	#prevReset := #rawReset;

END_FUNCTION_BLOCK

DATA_BLOCK "DB_RecipeProgram3"
{ S7_Optimized_Access := 'TRUE' }
VERSION : 0.1
NON_RETAIN
// -----------------------------------------------------------------------------
// DB_RecipeProgram3 - Recipe data for Program 3
// -----------------------------------------------------------------------------
   VAR
      Header : "RecipeHeader";
      Lines : Array[0..349] of "RecipeLine";
   END_VAR


BEGIN

END_DATA_BLOCK

DATA_BLOCK "DB_Manual"
{ S7_Optimized_Access := 'TRUE' }
VERSION : 0.3
NON_RETAIN
// -----------------------------------------------------------------------------
// DB_Manual - Manual mode control
// -----------------------------------------------------------------------------
   VAR
      ManualModeActive : Bool;
      SelectedAxis : Int;   // 0=X, 1=Z, 2=Tool, 3=Spindle
      ActiveAxis : Int;   // Currently active axis (-1 = none)
      JogSpeed : Real;   // mm/s
      JogIncrement : Real;   // mm per step
      HomingMode : Int;   // 0=Passive, 2=Active, 3=Active+Zero
      HomePosition : Real;   // Home position offset Jog buttons (both naming conventions)
      Btn_JogPlus : Bool;
      Btn_JogMinus : Bool;
      Jog_Plus : Bool;   // Alias
      Jog_Minus : Bool;   // Alias
      Btn_StepPlus : Bool;   // Incremental step +
      Btn_StepMinus : Bool;   // Incremental step - Homing buttons
      Btn_Home : Bool;
      Btn_HomeAxis : Bool;   // Alias for Btn_Home
      Btn_HomeAll : Bool;   // Home all axes
      Btn_GoSafe : Bool;
      Btn_GoZero : Bool;   // Absolute move
      MoveToPosition : Real;   // Target position
      Btn_MoveAbsolute : Bool;   // Execute move Tool step buttons
      Btn_ToolStepCW : Bool;   // Tool step clockwise
      Btn_ToolStepCCW : Bool;   // Tool step counter-clockwise
      ToolStepAngle : Real;   // Step angle (degrees)
      ToolStepSpeed : Real;   // Tool step velocity (deg/s)
      ToolPosition : Real;   // Current tool position (degrees) Spindle manual control
      Btn_SpindleStart : Bool;   // Start spindle
      Btn_SpindleStop : Bool;   // Stop spindle
      Btn_SpindleAckError : Bool;   // Acknowledge spindle error only (machine reset not required)
      Manual_SpindleSpeed : Real;   // Spindle speed (RPM)
      Manual_SpindleDir : Int;   // 1=CW, -1=CCW Status (multiple naming conventions for HMI compatibility)
      JogBusy : Bool;
      ManualBusy : Bool;   // Alias for JogBusy
      JogError : Bool;
      ManualError : Bool;   // Alias for JogError
      JogErrorID : Word;
      ManualErrorID : Word;   // Alias for JogErrorID Selected axis info (output)
      SelectedAxisName : String[20];
      SelectedAxisPos : Real;
      SelectedAxisHomed : Bool;
      SelectedAxisReady : Bool;   // =========================================================== CYLINDER MANUAL CONTROL One HMI screen controls all cylinders via SelectedCylinder. HMI writes to these fields; FC_CylinderDispatch routes to the correct DB_CylinderX instance each scan. To add a cylinder: add DB_CylinderN in 02_DataBlocks.scl, add OB1 calls, and add a CASE branch in FC_CylinderDispatch. ===========================================================
      SelectedCylinder : Int;   // Active cylinder (1..N)
      Btn_CylExtend : Bool;   // Extend command
      Btn_CylExtendFull : Bool;   // Full extend (ignore sensor)
      Btn_CylRetract : Bool;   // Retract command
      Btn_CylRetractFull : Bool;   // Full retract (bypass sensors, pulse use)
      Btn_CylGotoPos : Bool;   // Rising edge: go to target (Mode 2 = zone-pulse, Mode 3 = extend to level)
      Cyl_TargetPos : Real;   // [Modes 2+3] Target position (mm)
      Cyl_Tolerance : Real;   // [Mode 2] Tolerance written to cylinder DB on Btn_ApplyType press
      Btn_ApplyType : Bool;   // Rising edge: write SelCyl_SetType + Cyl_Tolerance â†’ cylinder DB
      SelCyl_SetType : Int;   // Desired PositioningMode (0â€“3) â€” HMI input field
      prevBtn_ApplyType : Bool;   // Edge detection (internal, not for HMI) Selected cylinder status (PLC â†’ HMI)
      SelCyl_Name : String[20];   // "Cylinder 1" etc.
      SelCyl_State : Int;   // State code
      SelCyl_StateText : String[14];   // State text
      SelCyl_AtSetpoint : Bool;   // Held at setpoint sensor
      SelCyl_AtRetract : Bool;   // At retract end
      SelCyl_AtTarget : Bool;   // Ruler mode: within Tolerance
      SelCyl_PosError : Real;   // Ruler mode: error = actual - target (mm)
      SelCyl_Error : Bool;   // Active error
      SelCyl_ErrorID : Word;   // Error code (16#05xx)
      SelCyl_ActualPos : Real;   // Current position (mm) from analog sensor
      SelCyl_Type : Int;   // Positioning mode: 0=Full stroke, 1=PNP sensor, 2=Linear ruler
      SelCyl_Toleranse : Real;   // Position tolerance (mm) - ruler mode only
      SelCyl_MaxPos : Real;   // Max allowed position (mm) - ruler mode only
      SelCyl_MinPos : Real;   // Min allowed position (mm) - ruler mode only
   END_VAR


BEGIN
   SelectedAxis := 0;
   ActiveAxis := -1;
   JogSpeed := 10.0;
   JogIncrement := 1.0;
   HomingMode := 3;
   HomePosition := 0.0;
   MoveToPosition := 0.0;
   ToolStepAngle := 90.0;
   ToolStepSpeed := 30.0;
   Manual_SpindleSpeed := 500.0;
   Manual_SpindleDir := 1;
   SelectedCylinder := 1;
   Cyl_TargetPos := 0.0;
   Cyl_Tolerance := 2.0;
   SelCyl_SetType := 0;

END_DATA_BLOCK

FUNCTION_BLOCK "FB_AlarmManager"
{ S7_Optimized_Access := 'TRUE' }
VERSION : 2.0
// -----------------------------------------------------------------------------
// FB_AlarmManager - Unified error management and monitoring
// DOC:
//  purpose: Single place to translate error codes to text, maintain active error state,
//           append to centralized DB_Error history, and provide outputs for monitoring.
//  inputs: NewError (rising edge), NewErrorCode, AcknowledgeError (edge)
//  outputs: HasActiveError, ActiveErrorCode, ActiveErrorText, ActiveSeverity, ActiveSource, ActiveTime
//  notes: Updates legacy DB_AlarmHistory for backward compatibility but centralizes storage in DB_Error.
// -----------------------------------------------------------------------------
   VAR_INPUT
      NewError : Bool;   // Rising edge triggers new active error
      NewErrorCode : Word;   // Numeric code describing error
      AcknowledgeError : Bool;   // Operator ack (edge)
      ActiveProgram : Int;   // ITEM-26: current recipe program (0=none); stored in alarm history
      ActiveLine : Int;   // ITEM-26: current recipe line (-1=outside recipe); stored in alarm history
   END_VAR

   VAR_OUTPUT
      HasActiveError : Bool;   // TRUE while an error is active (until ack)
      ActiveErrorCode : Word;   // Current active error code
      ActiveErrorText : String[80];   // Human readable text for HMI (English)
      ActiveErrorText_ES : String[80];   // Texto de error para HMI (EspaÃ±ol)
      ActiveSeverity : Byte;   // Priority tier: 1=warning, 2=project, 3=motion/TO, 4=safety (higher preempts lower on HMI display)
      ActiveSource : String[20];   // Source category string
      ActiveTime {InstructionName := 'DTL'; LibVersion := '1.0'} : DTL;   // Timestamp of active error
   END_VAR

   VAR
      prevNewError : Bool;   // previous NewError for edge detection
      currentTime {InstructionName := 'DTL'; LibVersion := '1.0'} : DTL;   // timestamp captured at NewError
      SystemTimeStatus : Int;   // RD_SYS_T return status
      i : Int;   // temporary loop index for history shift
      internalNewError : Bool;
      internalErrorCode : Word;
      fromQueue : Bool;   // TRUE when error came from DB_SystemEvents queue
      newHistCode : Word;   // new error code for history push (independent of first-error latch)
      newHistText : String[80];   // new error text for history push (independent of first-error latch)
      newHistSource : String[20];   // new error source for history push (independent of first-error latch)
      latchedText_ES : String[80];   // ES text of the DISPLAYED (latched) error -- DB_Error has no Details_ES field, so the Spanish counterpart is kept here for the secondary-error restore path (EN/ES must describe the same error)
   END_VAR


BEGIN

	#internalNewError := #NewError;
	#internalErrorCode := #NewErrorCode;
	#fromQueue := FALSE;

	// Dequeue one item per scan from DB_SystemEvents error ring buffer (written by FC_ReportError).
	// Processing one per scan is intentional: avoids two errors overwriting each other in the same
	// AlarmManager call. Any remaining items are consumed on subsequent scans.
	IF "DB_SystemEvents".EQ_Count > 0 THEN
	    #internalNewError := TRUE;
	    #internalErrorCode := "DB_SystemEvents".EQ_Code["DB_SystemEvents".EQ_Head];
	    "DB_Diagnostic".Error_Text := "DB_SystemEvents".EQ_Details["DB_SystemEvents".EQ_Head];
	    "DB_Diagnostic".Error_Code := "DB_SystemEvents".EQ_Code["DB_SystemEvents".EQ_Head];
	    "DB_SystemEvents".EQ_Head := ("DB_SystemEvents".EQ_Head + 1) MOD 4;
	    "DB_SystemEvents".EQ_Count := "DB_SystemEvents".EQ_Count - 1;
	    #fromQueue := TRUE;
	END_IF;

	// Handle new error
	// Queue path (fromQueue): always process â€” queue already guarantees one item per scan,
	//   so edge detection would drop consecutive errors when prevNewError stays TRUE.
	// Direct path (NewError input from FB_Process): edge-triggered to prevent repeated firing.
	IF #internalErrorCode <> 0 AND (#fromQueue OR (#internalNewError AND NOT #prevNewError)) THEN
	    #ActiveErrorCode := #internalErrorCode;
	    #SystemTimeStatus := RD_SYS_T(OUT => #currentTime);

	    // Translate code -> text
	    // CASE always runs for both paths to guarantee a Spanish translation.
	    // Queue path: EN is overridden after the CASE with the richer diagnostic text
	    //   from DB_Diagnostic.Error_Text (contains TO codes, line numbers).
	    //   ES remains from the CASE table -- proper Spanish, not English diagnostic text.
	    // Direct path: both EN and ES come from the CASE table only.
	    CASE #internalErrorCode OF
	            // Axis Movement Errors
	        16#0001:
	            #ActiveErrorText := 'X Axis: Move command failed';
	            #ActiveErrorText_ES := 'Eje X: fallo en comando de movimiento';
	        16#0002:
	            #ActiveErrorText := 'Z Axis: Move command failed';
	            #ActiveErrorText_ES := 'Eje Z: fallo en comando de movimiento';
	        16#0003:
	            #ActiveErrorText := 'X Axis: Homing failed';
	            #ActiveErrorText_ES := 'Eje X: fallo en referenciado';
	        16#0004:
	            #ActiveErrorText := 'Z Axis: Homing failed';
	            #ActiveErrorText_ES := 'Eje Z: fallo en referenciado';
	        16#0005:
	            #ActiveErrorText := 'Drive fault - check servo';
	            #ActiveErrorText_ES := 'Fallo en variador - revisar servo';
	        16#0006:
	            #ActiveErrorText := 'Tool Axis: Move failed';
	            #ActiveErrorText_ES := 'Eje herramienta: fallo de movimiento';
	        16#0007:
	            #ActiveErrorText := 'Tool Axis: Homing failed';
	            #ActiveErrorText_ES := 'Eje herramienta: fallo de referenciado';
	        16#0008:
	            #ActiveErrorText := 'Motion timeout - axis stuck';
	            #ActiveErrorText_ES := 'Tiempo de movimiento excedido - eje bloqueado';
	        16#0009:
	            #ActiveErrorText := 'X drive power failed';
	            #ActiveErrorText_ES := 'Fallo de potencia variador X';
	        16#000A:
	            #ActiveErrorText := 'Z drive power failed';
	            #ActiveErrorText_ES := 'Fallo de potencia variador Z';
	        16#000B:
	            #ActiveErrorText := 'Homing timeout - check ref switch';
	            #ActiveErrorText_ES := 'Tiempo de referenciado excedido - revisar sensor';
	        16#000C:
	            #ActiveErrorText := 'Drive ready timeout - check contactor/enable wiring';
	            #ActiveErrorText_ES := 'Tiempo de espera variador - revisar contactor/cableado';
	        16#000D:
	            #ActiveErrorText := 'Tool drive power failed';           // ITEM-29
	            #ActiveErrorText_ES := 'Fallo de potencia variador herramienta';
	        16#0012:
	            #ActiveErrorText := 'ToolHeadLock: extend timeout - check cylinder/sensor';
	            #ActiveErrorText_ES := 'Bloqueo cabezal: tiempo de extension excedido - revisar cilindro/sensor';
	        16#0010:
	            #ActiveErrorText := 'User pressed STOP';
	            #ActiveErrorText_ES := 'Operador presiono PARO';
	            // TO (Technology Object) fault poller (FB_Process, StatusBits.Error rising edge)
	        16#0021:
	            #ActiveErrorText := 'X axis TO fault - check TO diagnostics';
	            #ActiveErrorText_ES := 'Fallo TO eje X - revisar diagnostico TO';
	        16#0022:
	            #ActiveErrorText := 'Z axis TO fault - check TO diagnostics';
	            #ActiveErrorText_ES := 'Fallo TO eje Z - revisar diagnostico TO';
	        16#0023:
	            #ActiveErrorText := 'Tool axis TO fault - check TO diagnostics';
	            #ActiveErrorText_ES := 'Fallo TO eje herramienta - revisar diagnostico TO';
	        16#0024:
	            #ActiveErrorText := 'Spindle TO fault - check TO diagnostics';
	            #ActiveErrorText_ES := 'Fallo TO husillo - revisar diagnostico TO';
	            // Soft Limits
	        16#0101:
	            #ActiveErrorText := 'X beyond MIN soft limit';
	            #ActiveErrorText_ES := 'X fuera de limite minimo';
	        16#0102:
	            #ActiveErrorText := 'X beyond MAX soft limit';
	            #ActiveErrorText_ES := 'X fuera de limite maximo';
	        16#0103:
	            #ActiveErrorText := 'Z beyond MIN soft limit';
	            #ActiveErrorText_ES := 'Z fuera de limite minimo';
	        16#0104:
	            #ActiveErrorText := 'Z beyond MAX soft limit';
	            #ActiveErrorText_ES := 'Z fuera de limite maximo';
	            // PNP Proximity Zone Errors (auto mode only; homing and manual bypass these)
	        16#0121:
	            #ActiveErrorText := 'PNP zone: X axis MIN proximity';
	            #ActiveErrorText_ES := 'Zona PNP: proximidad MIN Eje X';
	        16#0122:
	            #ActiveErrorText := 'PNP zone: X axis MAX proximity';
	            #ActiveErrorText_ES := 'Zona PNP: proximidad MAX Eje X';
	        16#0123:
	            #ActiveErrorText := 'PNP zone: Z axis MIN proximity';
	            #ActiveErrorText_ES := 'Zona PNP: proximidad MIN Eje Z';
	        16#0124:
	            #ActiveErrorText := 'PNP zone: Z axis MAX proximity';
	            #ActiveErrorText_ES := 'Zona PNP: proximidad MAX Eje Z';
	            // Tool Errors
	        16#0201:
	            #ActiveErrorText := 'Invalid tool number';
	            #ActiveErrorText_ES := 'Numero de herramienta invalido';
	        16#0202:
	            #ActiveErrorText := 'Tool number out of range';
	            #ActiveErrorText_ES := 'Numero de herramienta fuera de rango';
	        16#0203:
	            #ActiveErrorText := 'Tool rotation timeout';
	            #ActiveErrorText_ES := 'Tiempo de rotacion herramienta excedido';
	        16#0204:
	            #ActiveErrorText := 'Retract to tool pos failed';
	            #ActiveErrorText_ES := 'Fallo al retraer a posicion de herramienta';
	        16#0205:
	            #ActiveErrorText := 'Tool rotation failed';
	            #ActiveErrorText_ES := 'Fallo en rotacion de herramienta';
	        16#0206:
	            #ActiveErrorText := 'Tool change timeout - check turret drive';
	            #ActiveErrorText_ES := 'Tiempo de cambio herramienta excedido - revisar variador';
	            // Recipe/G-code Errors
	        16#0301:
	            #ActiveErrorText := 'Recipe: Invalid command';
	            #ActiveErrorText_ES := 'Receta: Comando invalido';
	        16#0302:
	            #ActiveErrorText := 'Recipe: Parse error';
	            #ActiveErrorText_ES := 'Receta: Error de analisis';
	        16#0303:
	            #ActiveErrorText := 'Recipe: Empty program';
	            #ActiveErrorText_ES := 'Receta: Programa vacio';
	        16#0304:
	            #ActiveErrorText := 'Recipe: Line count zero';
	            #ActiveErrorText_ES := 'Receta: Conteo de lineas cero';
	        16#0305:
	            #ActiveErrorText := 'PreScan: Path exceeds limits';
	            #ActiveErrorText_ES := 'PreVerificacion: Trayectoria fuera de limites';
	        16#0306:
	            #ActiveErrorText := 'Recipe: Invalid feedrate';
	            #ActiveErrorText_ES := 'Receta: Avance invalido';
	        16#0307:
	            #ActiveErrorText := 'Recipe: Motion timeout';
	            #ActiveErrorText_ES := 'Receta: Tiempo de movimiento excedido';
	        16#0308:
	            #ActiveErrorText := 'Recipe: Invalid tool number';
	            #ActiveErrorText_ES := 'Receta: Numero de herramienta invalido';
	        16#0309:
	            #ActiveErrorText := 'BackSupport cylinder error - target not reached';
	            #ActiveErrorText_ES := 'Error cilindro BackSupport - posicion no alcanzada';
	        16#030A:
	            #ActiveErrorText := 'Spindle at-speed timeout (10s)';
	            #ActiveErrorText_ES := 'Husillo: tiempo de velocidad excedido (10s)';
	        16#030B:
	            #ActiveErrorText := 'Spindle stop timeout (15s)';
	            #ActiveErrorText_ES := 'Husillo: tiempo de paro excedido (15s)';
	        16#0310:
	            #ActiveErrorText := 'Recipe not loaded - check TotalLines';
	            #ActiveErrorText_ES := 'Receta no cargada - revisar TotalLines';
	            // Safety Errors
	        16#0401:
	            #ActiveErrorText := 'EMERGENCY STOP ACTIVE!';
	            #ActiveErrorText_ES := 'PARO DE EMERGENCIA ACTIVO!';
	        16#0402:
	            #ActiveErrorText := 'Safety door is open';
	            #ActiveErrorText_ES := 'Puerta de seguridad abierta';
	        16#0403:
	            #ActiveErrorText := 'Drives not ready';
	            #ActiveErrorText_ES := 'Variadores no listos';
	        16#0404:
	            #ActiveErrorText := 'Air pressure too low';
	            #ActiveErrorText_ES := 'Presion de aire baja';
	        16#0405:
	            #ActiveErrorText := 'Safety interlock active';
	            #ActiveErrorText_ES := 'Interlock de seguridad activo';
	        16#0406:
	            #ActiveErrorText := 'E-Stop contact discrepancy!';
	            #ActiveErrorText_ES := 'Discrepancia en contacto Paro de Emergencia!';
	            // Spindle Errors
	        16#0501:
	            #ActiveErrorText := 'Spindle: Power-on failed';
	            #ActiveErrorText_ES := 'Husillo: fallo al encender';
	        16#0502:
	            #ActiveErrorText := 'Spindle: Run command failed';
	            #ActiveErrorText_ES := 'Husillo: fallo al ejecutar comando';
	        16#0503:
	            #ActiveErrorText := 'Spindle: Halt failed';
	            #ActiveErrorText_ES := 'Husillo: fallo al detener';
	        16#0504:
	            #ActiveErrorText := 'Spindle: Speed not reached';
	            #ActiveErrorText_ES := 'Husillo: velocidad no alcanzada';
	        16#0505:
	            #ActiveErrorText := 'Spindle: Drive enable timeout';
	            #ActiveErrorText_ES := 'Husillo: tiempo de habilitacion excedido';
	            // NOTE: Siemens TO (Technology Object) error codes (16#8xxx) are NOT passed here
	            // directly. They are decoded via FC_TO_ErrorText and written to
	            // DB_Diagnostic.TO_ErrorText + DB_HMI.ErrorDetail at the point of failure.
	            // This CASE only handles project-level error codes (16#0001-16#05FF).
	        ELSE
	            #ActiveErrorText := 'Unknown error code';
	            #ActiveErrorText_ES := 'Codigo de error desconocido';
	    END_CASE;
	    // Queue path: override EN with the detailed diagnostic text (TO codes, line numbers);
	    // ES stays from CASE table above (proper Spanish translation).
	    IF #fromQueue THEN
	        #ActiveErrorText := "DB_Diagnostic".Error_Text;
	    END_IF;

	    // Severity & source mapping (explicit ranges)
	    // Priority tiers (higher tier preempts lower on the HMI display, see latch below):
	    //   4 = safety interlock (E-Stop, door, air, drives, HW limit)
	    //   3 = motion / TO fault (axis, homing, drive power, soft limit, PNP zone, tool motion, spindle)
	    //   2 = project error (recipe validation, tool configuration)
	    //   1 = warning / info (user stop, unknown codes)
	    IF #ActiveErrorCode >= 16#0400 AND #ActiveErrorCode < 16#0500 THEN
	        #ActiveSeverity := 4;
	        #ActiveSource := 'Safety';
	    ELSIF #ActiveErrorCode >= 16#0111 AND #ActiveErrorCode < 16#0120 THEN
	        #ActiveSeverity := 4;
	        #ActiveSource := 'HW Limit';
	    ELSIF #ActiveErrorCode >= 16#0121 AND #ActiveErrorCode < 16#0130 THEN
	        #ActiveSeverity := 3;
	        #ActiveSource := 'PNP Zone';  // PNP proximity zone errors (auto mode)
	    ELSIF #ActiveErrorCode = 16#0010 THEN
	        #ActiveSeverity := 1;
	        #ActiveSource := 'Operator';  // user STOP must never preempt a real fault
	    ELSIF #ActiveErrorCode >= 16#0001 AND #ActiveErrorCode <= 16#002F THEN
	        #ActiveSeverity := 3;
	        #ActiveSource := 'Axis';      // axis/homing/power, 16#0012 ToolHeadLock, 16#0021-0024 TO poller
	    ELSIF #ActiveErrorCode >= 16#0101 AND #ActiveErrorCode < 16#0110 THEN
	        #ActiveSeverity := 3;
	        #ActiveSource := 'Soft Limit';
	    ELSIF #ActiveErrorCode >= 16#0203 AND #ActiveErrorCode <= 16#0206 THEN
	        #ActiveSeverity := 3;
	        #ActiveSource := 'Tool';      // tool motion faults (rotation fail/timeout)
	    ELSIF #ActiveErrorCode >= 16#0200 AND #ActiveErrorCode < 16#0210 THEN
	        #ActiveSeverity := 2;
	        #ActiveSource := 'Tool';      // tool configuration (invalid/out of range)
	    ELSIF #ActiveErrorCode >= 16#0300 AND #ActiveErrorCode <= 16#0310 THEN
	        #ActiveSeverity := 2;
	        #ActiveSource := 'Recipe';    // <= includes 16#0310
	    ELSIF #ActiveErrorCode >= 16#0500 AND #ActiveErrorCode < 16#0510 THEN
	        #ActiveSeverity := 3;
	        #ActiveSource := 'Spindle';   // spindle motion faults
	    ELSE
	        #ActiveSeverity := 1;
	        #ActiveSource := 'Unknown';
	    END_IF;

	    // Save new error info for history before the latch guard may restore output vars
	    #newHistCode := #ActiveErrorCode;
	    #newHistText := #ActiveErrorText;
	    #newHistSource := #ActiveSource;

	    // Severity-priority latch: the display (DB_Error.Code, HMI text) shows the
	    // highest-severity error of the fault sequence. A new error replaces the displayed
	    // one only if its priority tier is STRICTLY higher (safety 4 > motion/TO 3 >
	    // project 2 > warning 1). Same or lower tier goes to history only, so the first
	    // error of a tier is never pushed aside by follow-up faults of the same tier
	    // (e.g. soft limit firing after the axis fault that caused it), while a TO/safety
	    // fault always wins the display over a project-level error that fired first.
	    // All errors always go to history. Cleared by AcknowledgeError.
	    IF NOT "DB_Error".Active OR (#ActiveSeverity > "DB_Error".Severity) THEN
	        #HasActiveError := TRUE;
	        #ActiveTime := #currentTime;
	        "DB_Error".Active := TRUE;
	        "DB_Error".Code := #ActiveErrorCode;
	        "DB_Error".Severity := #ActiveSeverity;
	        "DB_Error".Source := #ActiveSource;
	        IF "DB_Diagnostic".Recipe_CurrentLine >= 0 AND (#ActiveSource = 'Recipe') THEN
	            "DB_Error".Line := "DB_Diagnostic".Recipe_CurrentLine;
	        ELSE
	            "DB_Error".Line := -1;
	        END_IF;
	        "DB_Error".TimeStamp := #currentTime;
	        "DB_Error".Details := #ActiveErrorText;
	        #latchedText_ES := #ActiveErrorText_ES;  // keep ES of the displayed error (no Details_ES in DB_Error)
	    ELSE
	        // Same/lower-tier secondary error: restore output vars to the displayed error
	        // so DB_HMI.ErrorText and callers still see the highest-priority root cause.
	        // ES is restored from latchedText_ES so both languages describe the SAME error
	        // (the CASE above already overwrote ActiveErrorText_ES with the new error's text).
	        #ActiveErrorCode := "DB_Error".Code;
	        #ActiveErrorText := "DB_Error".Details;
	        #ActiveErrorText_ES := #latchedText_ES;
	        #ActiveSeverity := "DB_Error".Severity;
	        #ActiveSource := "DB_Error".Source;
	        #ActiveTime := "DB_Error".TimeStamp;
	        #HasActiveError := TRUE;
	    END_IF;
	    "DB_Error".TotalErrorCount := "DB_Error".TotalErrorCount + 1;
	    // History: always push the new error (not the latched first-error values)
	    FOR #i := 10 TO 2 BY -1 DO
	        "DB_Error".History_Code[#i] := "DB_Error".History_Code[#i - 1];
	        "DB_Error".History_Time[#i] := "DB_Error".History_Time[#i - 1];
	        "DB_Error".History_Source[#i] := "DB_Error".History_Source[#i - 1];
	        "DB_Error".History_Details[#i] := "DB_Error".History_Details[#i - 1];
	    END_FOR;
	    "DB_Error".History_Code[1] := #newHistCode;
	    "DB_Error".History_Time[1] := #currentTime;
	    "DB_Error".History_Source[1] := #newHistSource;
	    "DB_Error".History_Details[1] := #newHistText;
	    "DB_Error".History_Index := "DB_Error".History_Index + 1;
	    IF "DB_Error".History_Index > 10 THEN
	        "DB_Error".History_Index := 1;
	    END_IF;
	    IF "DB_Error".History_Count < 10 THEN
	        "DB_Error".History_Count := "DB_Error".History_Count + 1;
	    END_IF;

	    // ITEM-26: write to DB_AlarmHistory 20-entry ring buffer (always push new error)
	    // Use #currentTime already captured above (same scan, consistent timestamp)
	    IF "DB_AlarmHistory".Hist_Clear THEN
	        "DB_AlarmHistory".Hist_Head := 0;
	        "DB_AlarmHistory".Hist_Count := 0;
	        "DB_AlarmHistory".Hist_SeqNum := 0;
	        "DB_AlarmHistory".Hist_Clear := FALSE;
	    END_IF;
	    "DB_AlarmHistory".Hist_Log["DB_AlarmHistory".Hist_Head].Timestamp := #currentTime;
	    "DB_AlarmHistory".Hist_Log["DB_AlarmHistory".Hist_Head].ErrorCode := #newHistCode;
	    "DB_AlarmHistory".Hist_Log["DB_AlarmHistory".Hist_Head].ProgramNum := #ActiveProgram;
	    "DB_AlarmHistory".Hist_Log["DB_AlarmHistory".Hist_Head].LineNum := #ActiveLine;
	    "DB_AlarmHistory".Hist_Log["DB_AlarmHistory".Hist_Head].ErrorText := LEFT(IN := #newHistText, L := 40);
	    "DB_AlarmHistory".Hist_Head := ("DB_AlarmHistory".Hist_Head + 1) MOD 20;
	    "DB_AlarmHistory".Hist_SeqNum := "DB_AlarmHistory".Hist_SeqNum + 1;
	    IF "DB_AlarmHistory".Hist_Count < 20 THEN
	        "DB_AlarmHistory".Hist_Count := "DB_AlarmHistory".Hist_Count + 1;
	    END_IF;
	END_IF;

	// Latch previous new error for edge detection
	#prevNewError := #internalNewError;

	// Acknowledge handling: clear active state but retain history snapshot
	IF #AcknowledgeError THEN
	    #ActiveErrorCode := 0;
	    #HasActiveError := FALSE;
	    #ActiveErrorText := '';
	    #ActiveErrorText_ES := '';  // BUG FIX (2026-07-02): was never cleared -- stale Spanish
	    // error text kept mirroring to DB_HMI.ErrorText_ES after Ack
	    #latchedText_ES := '';
	    #ActiveSeverity := 0;
	    #ActiveSource := '';
	    #ActiveTime := DTL#1970-01-01-00:00:00;
	    // legacy DB_AlarmHistory removed; history retained in DB_Error
	    "DB_Error".Active := FALSE;
	    "DB_Error".Code := 0;  // BUG FIX: clear code so DB_HMI_Errors bits go FALSE
	    "DB_Error".Details := CONCAT(IN1 := "DB_Error".Details, IN2 := ' [ACK]');
	END_IF;

	// =========================================================================
	// DB_HMI_Errors - Pack error bits into Words for HMI Discrete Alarms
	// Word.Bit = one alarm line in HMI Alarm View
	// =========================================================================

	// AlarmWord_Axis: Bits 0-7
	"DB_HMI_Errors".AlarmWord_Axis :=
	BOOL_TO_WORD("DB_Error".Code = 16#0001) OR
	SHL(IN := BOOL_TO_WORD("DB_Error".Code = 16#0002), N := 1) OR
	SHL(IN := BOOL_TO_WORD("DB_Error".Code = 16#0003), N := 2) OR
	SHL(IN := BOOL_TO_WORD("DB_Error".Code = 16#0004), N := 3) OR
	SHL(IN := BOOL_TO_WORD("DB_Error".Code = 16#0005), N := 4) OR
	SHL(IN := BOOL_TO_WORD("DB_Error".Code = 16#0006), N := 5) OR
	SHL(IN := BOOL_TO_WORD("DB_Error".Code = 16#0007), N := 6) OR
	SHL(IN := BOOL_TO_WORD("DB_Error".Code = 16#0008), N := 7) OR
	SHL(IN := BOOL_TO_WORD("DB_Error".Code = 16#000D), N := 8);  // ITEM-29: tool drive power fault

	// AlarmWord_Limits: Bits 0-3 soft, 4-7 hardware
	"DB_HMI_Errors".AlarmWord_Limits :=
	BOOL_TO_WORD("DB_Error".Code = 16#0101) OR
	SHL(IN := BOOL_TO_WORD("DB_Error".Code = 16#0102), N := 1) OR
	SHL(IN := BOOL_TO_WORD("DB_Error".Code = 16#0103), N := 2) OR
	SHL(IN := BOOL_TO_WORD("DB_Error".Code = 16#0104), N := 3) OR
	SHL(IN := BOOL_TO_WORD("DB_Error".Code = 16#0111), N := 4) OR
	SHL(IN := BOOL_TO_WORD("DB_Error".Code = 16#0112), N := 5) OR
	SHL(IN := BOOL_TO_WORD("DB_Error".Code = 16#0113), N := 6) OR
	SHL(IN := BOOL_TO_WORD("DB_Error".Code = 16#0114), N := 7);

	// AlarmWord_Tool: Bits 0-4
	"DB_HMI_Errors".AlarmWord_Tool :=
	BOOL_TO_WORD("DB_Error".Code = 16#0201) OR
	SHL(IN := BOOL_TO_WORD("DB_Error".Code = 16#0202), N := 1) OR
	SHL(IN := BOOL_TO_WORD("DB_Error".Code = 16#0203), N := 2) OR
	SHL(IN := BOOL_TO_WORD("DB_Error".Code = 16#0204), N := 3) OR
	SHL(IN := BOOL_TO_WORD("DB_Error".Code = 16#0205), N := 4);

	// AlarmWord_Recipe: Bits 0-7
	"DB_HMI_Errors".AlarmWord_Recipe :=
	BOOL_TO_WORD("DB_Error".Code = 16#0301) OR
	SHL(IN := BOOL_TO_WORD("DB_Error".Code = 16#0302), N := 1) OR
	SHL(IN := BOOL_TO_WORD("DB_Error".Code = 16#0303), N := 2) OR
	SHL(IN := BOOL_TO_WORD("DB_Error".Code = 16#0304), N := 3) OR
	SHL(IN := BOOL_TO_WORD("DB_Error".Code = 16#0305), N := 4) OR
	SHL(IN := BOOL_TO_WORD("DB_Error".Code = 16#0306), N := 5) OR
	SHL(IN := BOOL_TO_WORD("DB_Error".Code = 16#0307), N := 6) OR
	SHL(IN := BOOL_TO_WORD("DB_Error".Code = 16#0308), N := 7);

	// AlarmWord_Safety: Bits 0-5
	"DB_HMI_Errors".AlarmWord_Safety :=
	BOOL_TO_WORD("DB_Error".Code = 16#0401) OR
	SHL(IN := BOOL_TO_WORD("DB_Error".Code = 16#0402), N := 1) OR
	SHL(IN := BOOL_TO_WORD("DB_Error".Code = 16#0403), N := 2) OR
	SHL(IN := BOOL_TO_WORD("DB_Error".Code = 16#0404), N := 3) OR
	SHL(IN := BOOL_TO_WORD("DB_Error".Code = 16#0405), N := 4) OR
	SHL(IN := BOOL_TO_WORD("DB_Error".Code = 16#0406), N := 5);

	// AlarmWord_Spindle: Bits 0-3
	"DB_HMI_Errors".AlarmWord_Spindle :=
	BOOL_TO_WORD("DB_Error".Code = 16#0501) OR
	SHL(IN := BOOL_TO_WORD("DB_Error".Code = 16#0502), N := 1) OR
	SHL(IN := BOOL_TO_WORD("DB_Error".Code = 16#0503), N := 2) OR
	SHL(IN := BOOL_TO_WORD("DB_Error".Code = 16#0504), N := 3);

	// AlarmWord_TO: Bits 0-4
	"DB_HMI_Errors".AlarmWord_TO :=
	BOOL_TO_WORD("DB_Error".Code = 16#8401) OR
	SHL(IN := BOOL_TO_WORD("DB_Error".Code = 16#8402), N := 1) OR
	SHL(IN := BOOL_TO_WORD("DB_Error".Code = 16#8403), N := 2) OR
	SHL(IN := BOOL_TO_WORD("DB_Error".Code = 16#8404), N := 3) OR
	SHL(IN := BOOL_TO_WORD("DB_Error".Code = 16#8405), N := 4);

	// Individual Bool flags (derived from DB_Error.Code)
	"DB_HMI_Errors".Err_X_MoveFailed := ("DB_Error".Code = 16#0001);
	"DB_HMI_Errors".Err_Z_MoveFailed := ("DB_Error".Code = 16#0002);
	"DB_HMI_Errors".Err_X_HomingFailed := ("DB_Error".Code = 16#0003);
	"DB_HMI_Errors".Err_Z_HomingFailed := ("DB_Error".Code = 16#0004);
	"DB_HMI_Errors".Err_DriveFault := ("DB_Error".Code = 16#0005);
	"DB_HMI_Errors".Err_ToolDrivePower := ("DB_Error".Code = 16#000D);  // ITEM-29
	"DB_HMI_Errors".Err_ToolMoveFailed := ("DB_Error".Code = 16#0006);
	"DB_HMI_Errors".Err_ToolHomingFailed := ("DB_Error".Code = 16#0007);
	"DB_HMI_Errors".Err_MotionTimeout := ("DB_Error".Code = 16#0008);
	"DB_HMI_Errors".Err_LockExtendTimeout := ("DB_Error".Code = 16#0012);
	"DB_HMI_Errors".Err_SoftLimit_X_Min := ("DB_Error".Code = 16#0101);
	"DB_HMI_Errors".Err_SoftLimit_X_Max := ("DB_Error".Code = 16#0102);
	"DB_HMI_Errors".Err_SoftLimit_Z_Min := ("DB_Error".Code = 16#0103);
	"DB_HMI_Errors".Err_SoftLimit_Z_Max := ("DB_Error".Code = 16#0104);
	"DB_HMI_Errors".Err_HWLimit_X_Min := ("DB_Error".Code = 16#0111);
	"DB_HMI_Errors".Err_HWLimit_X_Max := ("DB_Error".Code = 16#0112);
	"DB_HMI_Errors".Err_HWLimit_Z_Min := ("DB_Error".Code = 16#0113);
	"DB_HMI_Errors".Err_HWLimit_Z_Max := ("DB_Error".Code = 16#0114);
	"DB_HMI_Errors".Err_InvalidToolNum := ("DB_Error".Code = 16#0201);
	"DB_HMI_Errors".Err_ToolOutOfRange := ("DB_Error".Code = 16#0202);
	"DB_HMI_Errors".Err_ToolRotTimeout := ("DB_Error".Code = 16#0203);
	"DB_HMI_Errors".Err_ToolRetractFail := ("DB_Error".Code = 16#0204);
	"DB_HMI_Errors".Err_ToolRotFailed := ("DB_Error".Code = 16#0205);
	"DB_HMI_Errors".Err_Recipe_InvalidCmd := ("DB_Error".Code = 16#0301);
	"DB_HMI_Errors".Err_Recipe_ParseErr := ("DB_Error".Code = 16#0302);
	"DB_HMI_Errors".Err_Recipe_Empty := ("DB_Error".Code = 16#0303);
	"DB_HMI_Errors".Err_Recipe_NoLines := ("DB_Error".Code = 16#0304);
	"DB_HMI_Errors".Err_PreScan_Limits := ("DB_Error".Code = 16#0305);
	"DB_HMI_Errors".Err_Recipe_Feedrate := ("DB_Error".Code = 16#0306);
	"DB_HMI_Errors".Err_Recipe_Timeout := ("DB_Error".Code = 16#0307);
	"DB_HMI_Errors".Err_Recipe_ToolNum := ("DB_Error".Code = 16#0308);
	"DB_HMI_Errors".Err_EStop := ("DB_Error".Code = 16#0401);
	"DB_HMI_Errors".Err_EStop_Discrepancy := ("DB_Error".Code = 16#0406);
	"DB_HMI_Errors".Err_DoorOpen := ("DB_Error".Code = 16#0402);
	"DB_HMI_Errors".Err_DrivesNotReady := ("DB_Error".Code = 16#0403);
	"DB_HMI_Errors".Err_AirPressure := ("DB_Error".Code = 16#0404);
	"DB_HMI_Errors".Err_SafetyInterlock := ("DB_Error".Code = 16#0405);
	"DB_HMI_Errors".Err_Spindle_Power := ("DB_Error".Code = 16#0501);
	"DB_HMI_Errors".Err_Spindle_Run := ("DB_Error".Code = 16#0502);
	"DB_HMI_Errors".Err_Spindle_Halt := ("DB_Error".Code = 16#0503);
	"DB_HMI_Errors".Err_Spindle_Speed := ("DB_Error".Code = 16#0504);
	"DB_HMI_Errors".Err_TO_Position := ("DB_Error".Code = 16#8401);
	"DB_HMI_Errors".Err_TO_Velocity := ("DB_Error".Code = 16#8402);
	"DB_HMI_Errors".Err_TO_NotReady := ("DB_Error".Code = 16#8403);
	"DB_HMI_Errors".Err_TO_NotEnabled := ("DB_Error".Code = 16#8404);
	"DB_HMI_Errors".Err_TO_LimitExceeded := ("DB_Error".Code = 16#8405);

	// Summary flags (non-zero Word = category has error)
	"DB_HMI_Errors".AnyAxisError := ("DB_HMI_Errors".AlarmWord_Axis <> 0);
	"DB_HMI_Errors".AnyLimitError := ("DB_HMI_Errors".AlarmWord_Limits <> 0);
	"DB_HMI_Errors".AnyToolError := ("DB_HMI_Errors".AlarmWord_Tool <> 0);
	"DB_HMI_Errors".AnyRecipeError := ("DB_HMI_Errors".AlarmWord_Recipe <> 0);
	"DB_HMI_Errors".AnySafetyError := ("DB_HMI_Errors".AlarmWord_Safety <> 0);
	"DB_HMI_Errors".AnySpindleError := ("DB_HMI_Errors".AlarmWord_Spindle <> 0);
	"DB_HMI_Errors".AnyError := "DB_Error".Active;


END_FUNCTION_BLOCK

DATA_BLOCK "DB_RecipeProgram4"
{ S7_Optimized_Access := 'TRUE' }
VERSION : 0.1
NON_RETAIN
// -----------------------------------------------------------------------------
// DB_RecipeProgram4 - Recipe data for Program 4
// -----------------------------------------------------------------------------
   VAR
      Header : "RecipeHeader";
      Lines : Array[0..349] of "RecipeLine";
   END_VAR


BEGIN

END_DATA_BLOCK

FUNCTION_BLOCK "FB_EStopDualChannel"
{ S7_Optimized_Access := 'TRUE' }
VERSION : 1.1
// =============================================================================
// Version_Recipe - 08_Main_OB1.scl
// Main organization block - entry point for cyclic execution
// =============================================================================
// =============================================================================
// FB_EStopDualChannel -- Dual-channel emergency stop (E-Stop) monitoring
//
// Physical wiring:
//   Safety_Estop_Ch1 â†’ PLC DI  NC contact -- normally CLOSED (TRUE)
//   Safety_Estop_Ch2 â†’ PLC DI  NO contact -- normally OPEN   (FALSE)
//   Safety_Estop     â†’ Marker (%M), written by this FB
//
// Normal state (button not pressed):
//   NC=TRUE,  NO=FALSE  â†’  EStop_OK=TRUE  (machine may run)
//
// Emergency stop (button pressed):
//   NC=FALSE, NO=TRUE   â†’  EStop_OK=FALSE (controlled stop)
//
// Discrepancy (contact/wiring fault):
//   NC=TRUE,  NO=TRUE   â†’  EStop_OK=FALSE + DiscrepancyAlarm  (NO contact stuck)
//   NC=FALSE, NO=FALSE  â†’  EStop_OK=FALSE + DiscrepancyAlarm  (NC contact stuck)
//   In both cases the machine fails safe.
//
// Discrepancy alarm behavior:
//   If channels remain inconsistent for DiscrepancyTimeout, DiscrepancyAlarm is TRUE for one scan.
//   This alarm generates error code 16#0406 via FC_ReportError.
//   HMI: DB_HMI.EStop_Discrepancy + DB_HMI.EStop_Ch1_OK + DB_HMI.EStop_Ch2_OK
// =============================================================================
   VAR_INPUT
      Ch1_NC : Bool;   // NC contact -- normal: TRUE (closed)
      Ch2_NO : Bool;   // NO contact -- normal: FALSE (open)
      DiscrepancyTimeout : Time := T#500MS;   // Discrepancy debounce time
   END_VAR

   VAR_OUTPUT
      EStop_OK : Bool;   // TRUE = button not pressed = machine may run
      Discrepancy : Bool;   // TRUE = channels inconsistent = contact/wiring fault (instantaneous)
      DiscrepancyAlarm : Bool;   // TRUE = timeout exceeded â†’ generate alarm (rising edge)
   END_VAR

   VAR
      tonDiscrepancy {InstructionName := 'TON_TIME'; LibVersion := '1.0'} : TON_TIME;   // Discrepancy debounce timer
      prevTimerQ : Bool;   // Previous timer output for rising edge detection
   END_VAR


BEGIN

	// Safe state: NC closed (TRUE) AND NO open (FALSE)
	// E-Stop OK as long as neither channel breaks this condition
	#EStop_OK := #Ch1_NC AND NOT #Ch2_NO;

	// Discrepancy: channels must always be opposite (NCâ‰ NO)
	// When NC=NO (both TRUE or both FALSE) â†’ contact fault
	#Discrepancy := NOT (#Ch1_NC XOR #Ch2_NO);

	// Debounce: filter simultaneous switching delays
	#tonDiscrepancy(IN := #Discrepancy,
	                PT := #DiscrepancyTimeout);

	// Alarm: rising edge -- triggered once per discrepancy event
	#DiscrepancyAlarm := #tonDiscrepancy.Q AND NOT #prevTimerQ;
	#prevTimerQ := #tonDiscrepancy.Q;

END_FUNCTION_BLOCK

FUNCTION_BLOCK "FB_SafetyMonitor"
{ S7_Optimized_Access := 'TRUE' }
VERSION : 1.0
// -----------------------------------------------------------------------------
// FB_SafetyMonitor - Check E-Stop, Door, Air Pressure, Drives
// DOC:
//  purpose: Evaluate hardware safety inputs and bypass flags, produce SafeToRun/SafeToJog.
//  inputs: EStop_OK, Door_Closed, AirPressure_OK, DrivesReady and bypass flags.
//  outputs: SafeToRun (machine may start), SafeToJog (manual jog allowed), ErrorCode (if unsafe).
//  notes: Returns immediately on first fatal safety failure to minimize decision latency.
// -----------------------------------------------------------------------------
   VAR_INPUT
      EStop_OK : Bool;   // TRUE if E-stop circuit is OK (no emergency)
      Door_Closed : Bool;   // TRUE if safety door closed
      AirPressure_OK : Bool;   // TRUE if air pressure sufficient
      DrivesReady : Bool;   // TRUE if drives report ready Bypass flags (from HMI) used only for testing; production should disable
      Bypass_EStop : Bool;
      Bypass_Door : Bool;
      Bypass_AirPressure : Bool;
      Bypass_Drives : Bool;
   END_VAR

   VAR_OUTPUT
      SafeToRun : Bool;   // TRUE => allowed to start program execution
      SafeToJog : Bool;   // TRUE => manual jogging permitted
      ErrorCode : Word;   // Non-zero if unsafe (map to DB_ErrorCodes)
   END_VAR


BEGIN

	// Runs every scan. RETURNs on first failing condition -- priority order matters.
	// EStop and Drive fault disable both SafeToRun and SafeToJog (jogging also forbidden).
	// Door and air pressure only disable SafeToRun (manual jog still permitted).
	#ErrorCode := 0;
	IF NOT #EStop_OK AND NOT #Bypass_EStop THEN
	    // EMERGENCY STOP active -- all motion forbidden
	    #SafeToRun := FALSE;
	    #SafeToJog := FALSE;
	    #ErrorCode := 16#0401;
	    "DB_Diagnostic".Error_Text := 'Safety: EMERGENCY STOP active';
	    RETURN;
	END_IF;
	// Drive readiness is NOT checked here.
	// In STATE_STOPPED, contactors are physically blocked (modePermit=0), so drives can never
	// report ready before starting. Blocking SafeToRun/SafeToJog here creates a deadlock.
	// Drive enable is handled automatically in STATE_STARTING (tonDriveReady timeout).
	// Drive faults while running are caught by prevDriveFaultX/Z detection â†’ STATE_ERROR.
	#SafeToJog := TRUE;
	IF NOT #Door_Closed AND NOT #Bypass_Door THEN
	    // Safety door open -- auto run forbidden, manual jog allowed
	    #SafeToRun := FALSE;
	    #ErrorCode := 16#0402;
	    "DB_Diagnostic".Error_Text := 'Safety: Safety door is open';
	    RETURN;
	END_IF;
	IF NOT #AirPressure_OK AND NOT #Bypass_AirPressure THEN
	    // Air pressure insufficient -- pneumatic system will not operate
	    #SafeToRun := FALSE;
	    #ErrorCode := 16#0404;
	    "DB_Diagnostic".Error_Text := 'Safety: Air pressure too low';
	    RETURN;
	END_IF;
	#SafeToRun := TRUE;

END_FUNCTION_BLOCK

FUNCTION_BLOCK "FB_LimitMonitor"
{ S7_Optimized_Access := 'TRUE' }
VERSION : 1.0
// -----------------------------------------------------------------------------
// FB_LimitMonitor - Check soft and hard limits
// DOC:
//  purpose: Validate current axis positions against configured soft limits and hardware limit switches.
//  inputs: ActualPos_X/Z, Homed_X/Z, HW limit switches.
//  outputs: LimitError (TRUE if any violation), ErrorCode (first matching error code).
//  notes: Soft limits from DB_MachineConfig are used; hardware limit switches take precedence.
//         Soft limits are only checked for a HOMED axis (Homed_X/Z = StatusBits.HomingDone):
//         before homing the TO position is meaningless (0 after restart, stale after a run),
//         so comparing it against limits would produce false trips.
// -----------------------------------------------------------------------------
   VAR_INPUT
      ActualPos_X : Real;   // Current X position (mm)
      ActualPos_Z : Real;   // Current Z position (mm)
      Homed_X : Bool;   // X axis homed (StatusBits.HomingDone) -- soft limits checked only when TRUE
      Homed_Z : Bool;   // Z axis homed (StatusBits.HomingDone) -- soft limits checked only when TRUE NC limit switches: TRUE=closed=OK, FALSE=open=limit triggered Cable break also reads FALSE â†’ fail-safe behavior
      HW_NC_X_Min : Bool;   // NC switch: X min (FALSE = limit hit)
      HW_NC_X_Max : Bool;   // NC switch: X max (FALSE = limit hit)
      HW_NC_Z_Min : Bool;   // NC switch: Z min (FALSE = limit hit)
      HW_NC_Z_Max : Bool;   // NC switch: Z max (FALSE = limit hit) PNP NO proximity sensors: TRUE=target detected=entered limit zone Triggered BEFORE NC switch â†’ early warning + second safety layer
      HW_PNP_X_Min : Bool;   // PNP NO sensor: X min (TRUE = limit zone)
      HW_PNP_X_Max : Bool;   // PNP NO sensor: X max (TRUE = limit zone)
      HW_PNP_Z_Min : Bool;   // PNP NO sensor: Z min (TRUE = limit zone)
      HW_PNP_Z_Max : Bool;   // PNP NO sensor: Z max (TRUE = limit zone)
   END_VAR

   VAR_OUTPUT
      LimitError : Bool;   // TRUE if any soft/hard limit violated
      ErrorCode : Word;   // Specific error code for HMI/alarm
   END_VAR


BEGIN

	// Runs every scan. Soft limits are read from DB_MachineConfig.
	// Hardware limit switches take priority over soft limits (physical end stop).
	// ErrorCode shows the last triggered fault -- multiple can be active simultaneously.
	#LimitError := FALSE;
	#ErrorCode := 0;
	// --- Software (Soft) Limits ---
	// Only checked while the axis is homed: an un-homed axis has no valid position
	// reference, so soft limits cannot mean anything before the reference seek completes.
	IF #Homed_X THEN
	    IF #ActualPos_X < "DB_MachineConfig".SoftLimit_MinX THEN
	        #LimitError := TRUE;
	        #ErrorCode := 16#0101;
	        "DB_Diagnostic".Error_Text := 'Limit: X axis below minimum soft limit';
	    END_IF;
	    IF #ActualPos_X > "DB_MachineConfig".SoftLimit_MaxX THEN
	        #LimitError := TRUE;
	        #ErrorCode := 16#0102;
	        "DB_Diagnostic".Error_Text := 'Limit: X axis above maximum soft limit';
	    END_IF;
	END_IF;
	IF #Homed_Z THEN
	    IF #ActualPos_Z < "DB_MachineConfig".SoftLimit_MinZ THEN
	        #LimitError := TRUE;
	        #ErrorCode := 16#0103;
	        "DB_Diagnostic".Error_Text := 'Limit: Z axis below minimum soft limit';
	    END_IF;
	    IF #ActualPos_Z > "DB_MachineConfig".SoftLimit_MaxZ THEN
	        #LimitError := TRUE;
	        #ErrorCode := 16#0104;
	        "DB_Diagnostic".Error_Text := 'Limit: Z axis above maximum soft limit';
	    END_IF;
	END_IF;
	// --- Hardware Limit Switches ---
	// NC switches: the TO (Technology Object) is configured with these as HW limits.
	// The TO handles deceleration and stop directly -- no PLC action required.
	// Only E-Stop cuts contactor power; PLC does NOT raise LimitError on NC hits.
	//
	// PNP proximity sensors: handled separately in FB_Process (inline halt block).
	// In auto mode: PNP â†’ MC_Halt on triggered axis + STATE_ERROR (codes 16#0121-0124).
	// In homing and manual mode: PNP is bypassed (expected zone during reference seek / manual op).

END_FUNCTION_BLOCK

FUNCTION_BLOCK "FB_Axis_Power"
{ S7_Optimized_Access := 'TRUE' }
VERSION : 0.2
// =============================================================================
// FB_Axis_Power -- Drive power enable/disable
//
// Enable = TRUE  â†’ MC_Power called, drive enabled.
// Enable = FALSE â†’ MC_Power stopped, drive disabled.
// Status = TRUE  â†’ Drive ready and enabled.
// =============================================================================
   VAR_INPUT
      Enable : Bool;   // TRUE = enable drive
   END_VAR

   VAR_OUTPUT
      Status : Bool;   // TRUE = drive active and ready
      Error : Bool;   // Drive enable error
      ErrorID : Word;   // MC_Power TO error code -- for drive fault details
   END_VAR

   VAR_IN_OUT
      Axis {InstructionName := 'TO_PositioningAxis'; LibVersion := '8.0'} : TO_PositioningAxis;
   END_VAR

   VAR
      MC_Power_Instance {InstructionName := 'MC_Power'; LibVersion := '8.0'} : MC_Power;
   END_VAR


BEGIN

	#MC_Power_Instance(
	                   Axis := #Axis,
	                   Enable := #Enable,
	                   Status => #Status,
	                   Error => #Error,
	                   ErrorID => #ErrorID
	);

END_FUNCTION_BLOCK

FUNCTION "FC_TO_ErrorText" : String
{ S7_Optimized_Access := 'TRUE' }
VERSION : 1.0
// ---------------------------------------------------------------------------
// FC_TO_ErrorText -- Converts a Siemens TO (Technology Object) error code to a
// readable short string. All MC_ error outputs (MC_Home, MC_MoveAbsolute, etc.)
// return a 16-bit WORD; this FC converts it to String[20].
//
// Reference: TIA Portal Help â†’ S7-1200 Technology Objects â†’ ErrorIDs
// Full list: TIA Portal â†’ Online â†’ TO Diagnostics â†’ Error Description
//
// Usage:
//   detail := FC_TO_ErrorText(Code := fbMoveX.ErrorID);
//   â†’ 'FollowError', 'NotHomed', '+HWLimit', etc.
// ---------------------------------------------------------------------------
   VAR_INPUT
      Code : Word;   // TO error code from MC_ function block
   END_VAR


BEGIN

	// Siemens S7-1200/1500 TO motion error codes (most common)
	CASE #Code OF
	    16#0000:
	        #FC_TO_ErrorText := 'OK';
	        // State / command errors
	    16#8001:
	        #FC_TO_ErrorText := 'AxisDisabled';      // Axis is disabled
	    16#8002:
	        #FC_TO_ErrorText := 'CmdNotAccepted';    // Command rejected in current state
	    16#8003:
	        #FC_TO_ErrorText := 'HomingRequired';    // Homing must be done first
	    16#8004:
	        #FC_TO_ErrorText := 'AxisInError';       // Axis is in error state
	    16#8005:
	        #FC_TO_ErrorText := 'LimitedByCfg';      // Vel/acc limited by TO config
	    16#8010:
	        #FC_TO_ErrorText := 'NotHomed';          // Homing not done
	    16#8011:
	        #FC_TO_ErrorText := 'AxisBusy';          // Axis busy with another command
	    16#8012:
	        #FC_TO_ErrorText := 'HomingActive';      // Homing already in progress
	    16#8013:
	        #FC_TO_ErrorText := 'NotEnabled';        // MC_Power not enabled
	    16#8014:
	        #FC_TO_ErrorText := 'DriveNotReady';     // Drive not ready (STO active?)
	    16#8015:
	        #FC_TO_ErrorText := 'STOActive';         // Safe Torque Off active
	    16#8016:
	        #FC_TO_ErrorText := 'SafeStopActive';    // Safe Stop function active
	        // Config / parameter errors
	    16#8100:
	        #FC_TO_ErrorText := 'ConfigError';       // TO configuration error
	    16#8101:
	        #FC_TO_ErrorText := 'InvalidParam';      // Parameter out of TO range
	    16#8102:
	        #FC_TO_ErrorText := 'HomingModeErr';     // Homing mode not supported
	        // Velocity / acceleration errors
	    16#8200:
	        #FC_TO_ErrorText := 'VelTooHigh';        // Velocity exceeds TO limit
	    16#8201:
	        #FC_TO_ErrorText := 'AccTooHigh';        // Acceleration exceeds TO limit
	    16#8202:
	        #FC_TO_ErrorText := 'JerkTooHigh';       // Jerk exceeds TO limit
	        // Stop / emergency
	    16#8500:
	        #FC_TO_ErrorText := 'EmergencyStop';     // TO emergency stop
	    16#8501:
	        #FC_TO_ErrorText := 'PowerRemoved';      // Power removed (E-Stop?)
	    16#8502:
	        #FC_TO_ErrorText := 'ErrorStop';         // Error-triggered stop
	        // Limit switch errors
	    16#8600:
	        #FC_TO_ErrorText := '+SoftLimit';        // Positive soft limit exceeded
	    16#8601:
	        #FC_TO_ErrorText := '-SoftLimit';        // Negative soft limit exceeded
	    16#8602:
	        #FC_TO_ErrorText := '+HWLimit';          // Positive hardware limit switch
	    16#8603:
	        #FC_TO_ErrorText := '-HWLimit';          // Negative hardware limit switch
	    16#8604:
	        #FC_TO_ErrorText := 'DriveFault';        // Servo drive fault
	    16#8605:
	        #FC_TO_ErrorText := 'EncoderErr';        // Encoder error
	    16#8606:
	        #FC_TO_ErrorText := 'DriveCommsLost';    // Drive communication timeout
	        // Following / deviation errors
	    16#8A00:
	        #FC_TO_ErrorText := 'FollowError';       // Following error too large
	    16#8A01:
	        #FC_TO_ErrorText := 'PosDeviation';      // Position deviation exceeded
	    16#8A02:
	        #FC_TO_ErrorText := 'SpdDeviation';      // Speed deviation exceeded
	    16#8A03:
	        #FC_TO_ErrorText := 'TorqueLimited';     // Torque limit active
	    ELSE
	        // Unknown code -- use TIA Portal Online â†’ TO Diagnostics for details
	        #FC_TO_ErrorText := 'UnknownTO';
	END_CASE;

END_FUNCTION

DATA_BLOCK "DB_RecipeProgram1"
{ S7_Optimized_Access := 'TRUE' }
VERSION : 0.1
NON_RETAIN
// =============================================================================
// 02b_RecipePrograms.scl
// Recipe program data blocks (DB_RecipeProgram1..5)
// Kept separate from 02_DataBlocks.scl so real recipe data is not overwritten
// when 02_DataBlocks.scl is regenerated.
// Depends on: 01_DataTypes.scl (RecipeHeader, RecipeLine UDTs)
// =============================================================================
// -----------------------------------------------------------------------------
// DB_RecipeProgram1 - Recipe data for Program 1
// -----------------------------------------------------------------------------
   VAR
      Header : "RecipeHeader";   // Program name, LineCount, Valid, bounding box
      Lines : Array[0..349] of "RecipeLine";   // 200 lines max
   END_VAR


BEGIN

END_DATA_BLOCK

